Yaskawa INFORM job: A_ROOF_SIDE_0617_2_PAINT_21.JBI

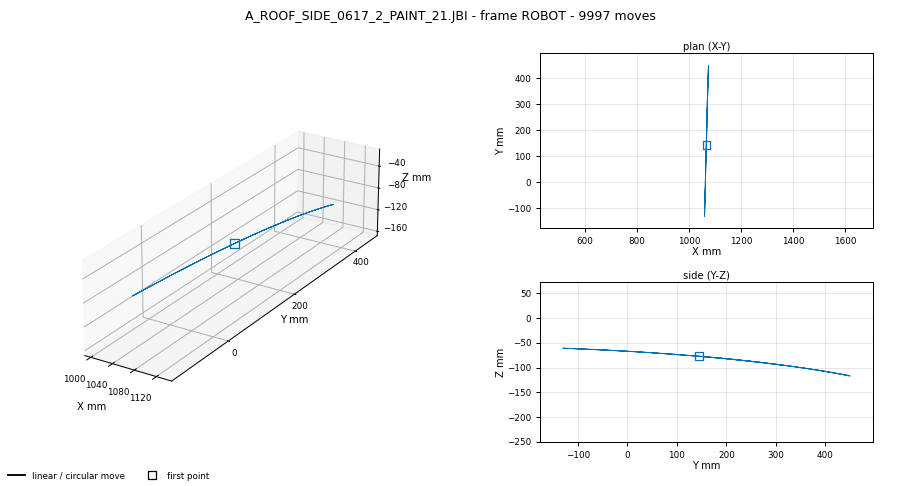
[picture p0: tool path of A_ROOF_SIDE_0617_2_PAINT_21.JBI in frame ROBOT, 9997 of 9997 moves have a stored position in this frame; points joined in program order, loops and branches not executed]
/JOB
//NAME A_ROOF_SIDE_0617_2_PAINT21
//POS
///NPOS 9997,0,0,0,0,0
///TOOL 1
///USER 0
///POSTYPE ROBOT
///RECTAN
///RCONF 1,0,0,0,0,0,0,0,0,0,0,0,0,0,0,0,0,0,0,0,0,0,0,0
C00000=1068.120,143.960,-76.437,172.975,27.840,155.057
C00001=1068.127,144.208,-76.458,172.976,27.843,155.058
C00002=1068.132,144.458,-76.479,172.978,27.845,155.058
C00003=1068.138,144.707,-76.500,172.981,27.848,155.058
C00004=1068.143,144.956,-76.521,172.982,27.851,155.059
C00005=1068.149,145.204,-76.542,172.984,27.854,155.059
C00006=1068.155,145.454,-76.563,172.985,27.857,155.059
C00007=1068.161,145.702,-76.584,172.988,27.860,155.060
C00008=1068.167,145.952,-76.605,172.989,27.862,155.060
C00009=1068.173,146.201,-76.626,172.991,27.865,155.061
C00010=1068.178,146.451,-76.647,172.992,27.868,155.061
C00011=1068.184,146.699,-76.668,172.995,27.870,155.061
C00012=1068.189,146.948,-76.689,172.996,27.873,155.062
C00013=1068.195,147.197,-76.710,172.998,27.876,155.062
C00014=1068.201,147.446,-76.730,172.999,27.879,155.063
C00015=1068.208,147.695,-76.752,173.001,27.881,155.063
C00016=1068.213,147.944,-76.773,173.003,27.885,155.063
C00017=1068.219,148.194,-76.794,173.005,27.887,155.064
C00018=1068.225,148.442,-76.816,173.007,27.890,155.064
C00019=1068.230,148.692,-76.836,173.008,27.893,155.065
C00020=1068.236,148.941,-76.858,173.011,27.896,155.065
C00021=1068.242,149.189,-76.879,173.012,27.898,155.065
C00022=1068.247,149.439,-76.900,173.014,27.901,155.066
C00023=1068.253,149.687,-76.921,173.015,27.904,155.066
C00024=1068.259,149.937,-76.943,173.018,27.907,155.066
C00025=1068.264,150.186,-76.963,173.019,27.909,155.067
C00026=1068.271,150.435,-76.985,173.021,27.912,155.067
C00027=1068.276,150.683,-77.006,173.022,27.915,155.068
C00028=1068.282,150.933,-77.028,173.025,27.918,155.068
C00029=1068.288,151.182,-77.048,173.026,27.921,155.068
C00030=1068.294,151.431,-77.070,173.028,27.923,155.069
C00031=1068.299,151.680,-77.092,173.030,27.926,155.069
C00032=1068.304,151.930,-77.113,173.032,27.929,155.070
C00033=1068.310,152.178,-77.134,173.034,27.932,155.070
C00034=1068.316,152.427,-77.156,173.035,27.935,155.070
C00035=1068.322,152.676,-77.177,173.038,27.938,155.071
C00036=1068.328,152.925,-77.199,173.039,27.940,155.071
C00037=1068.333,153.174,-77.219,173.041,27.943,155.071
C00038=1068.339,153.423,-77.241,173.042,27.945,155.072
C00039=1068.345,153.672,-77.262,173.045,27.948,155.072
C00040=1068.351,153.921,-77.284,173.046,27.951,155.073
C00041=1068.356,154.170,-77.306,173.048,27.954,155.073
C00042=1068.362,154.419,-77.327,173.049,27.957,155.074
C00043=1068.367,154.668,-77.348,173.052,27.960,155.074
C00044=1068.373,154.917,-77.369,173.053,27.962,155.074
C00045=1068.379,155.166,-77.391,173.055,27.965,155.075
C00046=1068.385,155.415,-77.412,173.058,27.968,155.075
C00047=1068.391,155.664,-77.434,173.059,27.971,155.075
C00048=1068.396,155.913,-77.456,173.061,27.974,155.076
C00049=1068.402,156.162,-77.478,173.062,27.976,155.076
C00050=1068.408,156.411,-77.499,173.065,27.979,155.077
C00051=1068.414,156.660,-77.520,173.066,27.982,155.077
C00052=1068.420,156.909,-77.542,173.068,27.985,155.078
C00053=1068.425,157.158,-77.564,173.070,27.988,155.078
C00054=1068.430,157.407,-77.584,173.072,27.990,155.078
C00055=1068.436,157.656,-77.606,173.073,27.993,155.079
C00056=1068.442,157.905,-77.627,173.076,27.996,155.079
C00057=1068.447,158.154,-77.650,173.077,27.999,155.079
C00058=1068.454,158.404,-77.671,173.079,28.001,155.080
C00059=1068.460,158.686,-77.696,173.081,28.005,155.080
C00060=1068.467,158.968,-77.721,173.083,28.008,155.081
C00061=1068.474,159.252,-77.745,173.085,28.011,155.081
C00062=1068.479,159.535,-77.770,173.088,28.014,155.082
C00063=1068.485,159.783,-77.792,173.089,28.017,155.082
C00064=1068.491,160.033,-77.813,173.091,28.020,155.082
C00065=1068.497,160.282,-77.835,173.094,28.023,155.083
C00066=1068.502,160.531,-77.857,173.095,28.025,155.083
C00067=1068.508,160.780,-77.878,173.097,28.028,155.084
C00068=1068.514,161.029,-77.900,173.099,28.031,155.084
C00069=1068.519,161.278,-77.922,173.101,28.034,155.084
C00070=1068.526,161.526,-77.944,173.102,28.037,155.085
C00071=1068.531,161.775,-77.966,173.104,28.039,155.085
C00072=1068.537,162.024,-77.988,173.106,28.042,155.086
C00073=1068.542,162.274,-78.010,173.108,28.045,155.086
C00074=1068.548,162.522,-78.031,173.109,28.048,155.086
C00075=1068.553,162.771,-78.054,173.112,28.051,155.087
C00076=1068.558,163.020,-78.076,173.113,28.054,155.087
C00077=1068.564,163.269,-78.098,173.115,28.057,155.088
C00078=1068.569,163.518,-78.120,173.117,28.060,155.088
C00079=1068.575,163.767,-78.141,173.119,28.063,155.088
C00080=1068.581,164.016,-78.164,173.121,28.065,155.089
C00081=1068.586,164.265,-78.186,173.123,28.068,155.089
C00082=1068.592,164.514,-78.208,173.125,28.071,155.090
C00083=1068.598,164.764,-78.230,173.126,28.074,155.090
C00084=1068.603,165.012,-78.252,173.129,28.077,155.090
C00085=1068.609,165.261,-78.274,173.130,28.080,155.091
C00086=1068.614,165.510,-78.296,173.132,28.083,155.091
C00087=1068.620,165.759,-78.318,173.134,28.086,155.092
C00088=1068.626,166.008,-78.340,173.136,28.089,155.092
C00089=1068.630,166.257,-78.362,173.138,28.092,155.093
C00090=1068.637,166.506,-78.385,173.140,28.094,155.093
C00091=1068.642,166.755,-78.407,173.141,28.097,155.093
C00092=1068.647,167.004,-78.429,173.144,28.100,155.094
C00093=1068.654,167.252,-78.451,173.145,28.103,155.094
C00094=1068.659,167.502,-78.473,173.147,28.106,155.095
C00095=1068.664,167.750,-78.496,173.150,28.109,155.095
C00096=1068.670,167.999,-78.518,173.151,28.112,155.096
C00097=1068.676,168.249,-78.540,173.153,28.115,155.096
C00098=1068.682,168.498,-78.562,173.155,28.118,155.096
C00099=1068.687,168.746,-78.584,173.157,28.120,155.097
C00100=1068.693,168.995,-78.607,173.159,28.123,155.097
C00101=1068.699,169.244,-78.629,173.161,28.126,155.098
C00102=1068.704,169.493,-78.651,173.162,28.129,155.098
C00103=1068.709,169.742,-78.673,173.165,28.132,155.098
C00104=1068.715,169.991,-78.696,173.166,28.135,155.099
C00105=1068.721,170.240,-78.718,173.168,28.137,155.099
C00106=1068.726,170.488,-78.741,173.170,28.140,155.100
C00107=1068.732,170.738,-78.763,173.172,28.143,155.100
C00108=1068.738,170.987,-78.785,173.175,28.146,155.100
C00109=1068.744,171.236,-78.807,173.176,28.149,155.101
C00110=1068.750,171.485,-78.830,173.178,28.151,155.101
C00111=1068.755,171.733,-78.852,173.180,28.155,155.102
C00112=1068.761,171.982,-78.875,173.182,28.158,155.102
C00113=1068.766,172.232,-78.897,173.184,28.161,155.102
C00114=1068.772,172.481,-78.920,173.186,28.163,155.103
C00115=1068.778,172.730,-78.941,173.187,28.166,155.103
C00116=1068.783,172.978,-78.964,173.190,28.169,155.104
C00117=1068.789,173.227,-78.987,173.191,28.172,155.104
C00118=1068.795,173.476,-79.009,173.194,28.175,155.104
C00119=1068.801,173.725,-79.031,173.195,28.178,155.105
C00120=1068.807,173.974,-79.054,173.197,28.180,155.105
C00121=1068.811,174.223,-79.076,173.200,28.183,155.106
C00122=1068.818,174.471,-79.099,173.201,28.186,155.106
C00123=1068.825,174.755,-79.125,173.204,28.190,155.107
C00124=1068.831,175.037,-79.150,173.206,28.193,155.107
C00125=1068.837,175.319,-79.175,173.208,28.196,155.107
C00126=1068.844,175.602,-79.201,173.210,28.199,155.108
C00127=1068.850,175.851,-79.224,173.213,28.202,155.108
C00128=1068.856,176.100,-79.246,173.214,28.205,155.109
C00129=1068.861,176.348,-79.269,173.217,28.208,155.109
C00130=1068.867,176.597,-79.292,173.218,28.210,155.109
C00131=1068.872,176.846,-79.314,173.220,28.213,155.110
C00132=1068.878,177.095,-79.336,173.222,28.216,155.110
C00133=1068.884,177.344,-79.359,173.224,28.219,155.111
C00134=1068.890,177.593,-79.382,173.226,28.222,155.111
C00135=1068.896,177.842,-79.405,173.228,28.225,155.112
C00136=1068.902,178.091,-79.427,173.230,28.228,155.112
C00137=1068.908,178.340,-79.450,173.232,28.231,155.112
C00138=1068.913,178.589,-79.472,173.235,28.234,155.113
C00139=1068.919,178.838,-79.495,173.236,28.236,155.113
C00140=1068.925,179.087,-79.518,173.239,28.239,155.113
C00141=1068.931,179.336,-79.541,173.240,28.242,155.114
C00142=1068.937,179.584,-79.564,173.242,28.245,155.114
C00143=1068.942,179.834,-79.586,173.244,28.248,155.115
C00144=1068.948,180.083,-79.609,173.246,28.251,155.115
C00145=1068.954,180.332,-79.632,173.248,28.254,155.115
C00146=1068.960,180.580,-79.654,173.250,28.256,155.116
C00147=1068.966,180.829,-79.677,173.252,28.259,155.116
C00148=1068.972,181.078,-79.700,173.254,28.262,155.117
C00149=1068.978,181.327,-79.723,173.257,28.265,155.117
C00150=1068.983,181.576,-79.746,173.258,28.268,155.117
C00151=1068.989,181.825,-79.769,173.261,28.271,155.118
C00152=1068.995,182.073,-79.791,173.262,28.273,155.118
C00153=1069.001,182.322,-79.814,173.265,28.276,155.119
C00154=1069.007,182.571,-79.837,173.266,28.279,155.119
C00155=1069.013,182.820,-79.860,173.269,28.282,155.119
C00156=1069.018,183.069,-79.883,173.270,28.285,155.120
C00157=1069.024,183.318,-79.906,173.273,28.288,155.120
C00158=1069.031,183.566,-79.928,173.275,28.290,155.121
C00159=1069.036,183.815,-79.951,173.277,28.293,155.121
C00160=1069.042,184.064,-79.974,173.279,28.296,155.121
C00161=1069.048,184.313,-79.997,173.281,28.299,155.122
C00162=1069.053,184.562,-80.020,173.283,28.302,155.122
C00163=1069.059,184.811,-80.043,173.285,28.305,155.123
C00164=1069.065,185.060,-80.066,173.287,28.307,155.123
C00165=1069.071,185.309,-80.089,173.289,28.310,155.123
C00166=1069.076,185.557,-80.113,173.291,28.314,155.124
C00167=1069.082,185.806,-80.136,173.293,28.317,155.124
C00168=1069.087,186.055,-80.159,173.295,28.319,155.125
C00169=1069.092,186.304,-80.183,173.298,28.322,155.125
C00170=1069.098,186.553,-80.206,173.299,28.326,155.126
C00171=1069.104,186.802,-80.229,173.302,28.329,155.126
C00172=1069.110,187.050,-80.252,173.303,28.331,155.126
C00173=1069.115,187.300,-80.276,173.306,28.335,155.127
C00174=1069.121,187.548,-80.299,173.307,28.338,155.127
C00175=1069.126,187.797,-80.322,173.310,28.341,155.128
C00176=1069.132,188.046,-80.346,173.311,28.343,155.128
C00177=1069.137,188.295,-80.369,173.314,28.347,155.129
C00178=1069.143,188.544,-80.392,173.315,28.350,155.129
C00179=1069.148,188.793,-80.415,173.318,28.352,155.130
C00180=1069.154,189.041,-80.439,173.319,28.355,155.130
C00181=1069.160,189.290,-80.462,173.322,28.359,155.130
C00182=1069.165,189.539,-80.485,173.324,28.362,155.131
C00183=1069.171,189.788,-80.509,173.326,28.364,155.131
C00184=1069.177,190.037,-80.532,173.329,28.367,155.132
C00185=1069.182,190.286,-80.556,173.330,28.371,155.132
C00186=1069.188,190.535,-80.580,173.333,28.374,155.133
C00187=1069.195,190.816,-80.606,173.335,28.377,155.133
C00188=1069.201,191.098,-80.632,173.337,28.380,155.134
C00189=1069.207,191.381,-80.660,173.339,28.384,155.134
C00190=1069.213,191.663,-80.686,173.342,28.387,155.134
C00191=1069.219,191.912,-80.709,173.344,28.390,155.135
C00192=1069.226,192.161,-80.733,173.346,28.393,155.135
C00193=1069.231,192.410,-80.757,173.348,28.396,155.136
C00194=1069.236,192.659,-80.780,173.351,28.399,155.136
C00195=1069.242,192.907,-80.804,173.352,28.402,155.137
C00196=1069.247,193.156,-80.827,173.355,28.405,155.137
C00197=1069.254,193.405,-80.850,173.356,28.408,155.137
C00198=1069.259,193.654,-80.874,173.359,28.411,155.138
C00199=1069.265,193.903,-80.898,173.360,28.414,155.138
C00200=1069.271,194.152,-80.921,173.363,28.417,155.139
C00201=1069.276,194.400,-80.945,173.365,28.420,155.139
C00202=1069.282,194.649,-80.968,173.367,28.423,155.140
C00203=1069.287,194.898,-80.992,173.370,28.426,155.140
C00204=1069.293,195.146,-81.016,173.371,28.429,155.141
C00205=1069.300,195.396,-81.039,173.374,28.432,155.141
C00206=1069.305,195.644,-81.064,173.376,28.435,155.141
C00207=1069.311,195.893,-81.087,173.378,28.438,155.142
C00208=1069.316,196.142,-81.111,173.380,28.441,155.142
C00209=1069.322,196.391,-81.134,173.382,28.444,155.143
C00210=1069.328,196.640,-81.158,173.384,28.447,155.143
C00211=1069.334,196.888,-81.182,173.387,28.450,155.144
C00212=1069.339,197.137,-81.205,173.388,28.453,155.144
C00213=1069.345,197.386,-81.230,173.391,28.456,155.144
C00214=1069.351,197.635,-81.253,173.393,28.459,155.145
C00215=1069.356,197.884,-81.277,173.395,28.462,155.145
C00216=1069.362,198.132,-81.300,173.398,28.465,155.146
C00217=1069.368,198.381,-81.325,173.399,28.468,155.146
C00218=1069.374,198.630,-81.349,173.402,28.471,155.147
C00219=1069.380,198.879,-81.372,173.403,28.474,155.147
C00220=1069.385,199.127,-81.396,173.406,28.477,155.147
C00221=1069.392,199.376,-81.420,173.408,28.481,155.148
C00222=1069.397,199.625,-81.444,173.410,28.483,155.148
C00223=1069.403,199.874,-81.467,173.412,28.486,155.149
C00224=1069.409,200.123,-81.492,173.415,28.489,155.149
C00225=1069.415,200.371,-81.515,173.416,28.492,155.150
C00226=1069.420,200.620,-81.540,173.419,28.495,155.150
C00227=1069.426,200.869,-81.563,173.422,28.498,155.150
C00228=1069.432,201.118,-81.587,173.423,28.501,155.151
C00229=1069.438,201.366,-81.611,173.426,28.504,155.151
C00230=1069.444,201.616,-81.636,173.428,28.507,155.152
C00231=1069.450,201.864,-81.659,173.430,28.510,155.152
C00232=1069.455,202.112,-81.683,173.432,28.513,155.152
C00233=1069.461,202.362,-81.707,173.434,28.516,155.153
C00234=1069.467,202.611,-81.731,173.436,28.519,155.153
C00235=1069.472,202.859,-81.755,173.439,28.523,155.154
C00236=1069.479,203.108,-81.779,173.441,28.525,155.154
C00237=1069.484,203.357,-81.804,173.443,28.528,155.155
C00238=1069.489,203.605,-81.828,173.446,28.532,155.155
C00239=1069.494,203.826,-81.850,173.447,28.535,155.156
C00240=1069.500,204.046,-81.871,173.449,28.537,155.156
C00241=1069.504,204.268,-81.892,173.451,28.540,155.156
C00242=1069.509,204.488,-81.914,173.453,28.543,155.157
C00243=1069.514,204.709,-81.935,173.455,28.546,155.157
C00244=1069.520,204.929,-81.957,173.457,28.549,155.158
C00245=1069.525,205.150,-81.978,173.459,28.551,155.158
C00246=1069.530,205.371,-82.000,173.461,28.554,155.158
C00247=1069.535,205.619,-82.024,173.463,28.557,155.159
C00248=1069.542,205.868,-82.048,173.465,28.560,155.159
C00249=1069.547,206.117,-82.073,173.468,28.563,155.160
C00250=1069.553,206.366,-82.097,173.469,28.566,155.160
C00251=1069.581,207.634,-82.221,173.612,28.641,155.164
C00252=1069.587,207.847,-82.243,173.614,28.644,155.164
C00253=1069.592,208.061,-82.265,173.616,28.648,155.165
C00254=1069.598,208.275,-82.286,173.618,28.651,155.165
C00255=1069.602,208.489,-82.308,173.619,28.655,155.166
C00256=1069.608,208.703,-82.329,173.621,28.658,155.167
C00257=1069.612,208.917,-82.351,173.622,28.662,155.167
C00258=1069.617,209.131,-82.373,173.625,28.665,155.168
C00259=1069.623,209.344,-82.394,173.626,28.668,155.168
C00260=1069.629,209.593,-82.419,173.629,28.673,155.169
C00261=1069.634,209.841,-82.444,173.630,28.677,155.170
C00262=1069.640,210.090,-82.469,173.633,28.681,155.170
C00263=1069.646,210.339,-82.495,173.634,28.685,155.171
C00264=1069.652,210.588,-82.520,173.636,28.689,155.171
C00265=1069.658,210.836,-82.545,173.639,28.693,155.172
C00266=1069.664,211.084,-82.570,173.640,28.697,155.173
C00267=1069.670,211.334,-82.595,173.643,28.701,155.173
C00268=1069.675,211.583,-82.621,173.644,28.705,155.174
C00269=1069.681,211.831,-82.646,173.647,28.709,155.175
C00270=1069.687,212.079,-82.671,173.649,28.713,155.175
C00271=1069.693,212.328,-82.697,173.650,28.717,155.176
C00272=1069.699,212.576,-82.722,173.653,28.721,155.177
C00273=1069.705,212.825,-82.748,173.654,28.725,155.178
C00274=1069.711,213.074,-82.773,173.657,28.729,155.178
C00275=1069.717,213.322,-82.798,173.659,28.733,155.179
C00276=1069.722,213.571,-82.824,173.661,28.737,155.179
C00277=1069.728,213.820,-82.849,173.663,28.741,155.180
C00278=1069.735,214.068,-82.875,173.665,28.745,155.181
C00279=1069.739,214.317,-82.900,173.667,28.749,155.181
C00280=1069.746,214.565,-82.926,173.669,28.753,155.182
C00281=1069.752,214.814,-82.951,173.671,28.757,155.183
C00282=1069.757,215.063,-82.977,173.673,28.761,155.183
C00283=1069.764,215.312,-83.002,173.676,28.765,155.184
C00284=1069.769,215.561,-83.028,173.677,28.769,155.185
C00285=1069.775,215.809,-83.053,173.679,28.773,155.185
C00286=1069.781,216.057,-83.078,173.682,28.777,155.186
C00287=1069.786,216.306,-83.104,173.683,28.781,155.187
C00288=1069.792,216.555,-83.130,173.686,28.785,155.187
C00289=1069.799,216.804,-83.155,173.687,28.789,155.188
C00290=1069.804,217.053,-83.181,173.690,28.793,155.189
C00291=1069.810,217.301,-83.206,173.692,28.797,155.189
C00292=1069.815,217.550,-83.232,173.694,28.801,155.190
C00293=1069.822,217.798,-83.258,173.696,28.805,155.191
C00294=1069.828,218.046,-83.283,173.698,28.809,155.191
C00295=1069.833,218.295,-83.309,173.700,28.813,155.192
C00296=1069.840,218.544,-83.335,173.702,28.817,155.193
C00297=1069.845,218.793,-83.361,173.705,28.821,155.193
C00298=1069.852,219.041,-83.387,173.706,28.825,155.194
C00299=1069.857,219.290,-83.413,173.709,28.829,155.195
C00300=1069.863,219.539,-83.438,173.711,28.833,155.195
C00301=1069.869,219.787,-83.463,173.713,28.837,155.196
C00302=1069.875,220.036,-83.490,173.715,28.841,155.197
C00303=1069.881,220.284,-83.515,173.717,28.845,155.197
C00304=1069.887,220.533,-83.541,173.719,28.849,155.198
C00305=1069.893,220.782,-83.566,173.721,28.853,155.199
C00306=1069.899,221.030,-83.593,173.724,28.857,155.199
C00307=1069.905,221.279,-83.618,173.725,28.861,155.200
C00308=1069.910,221.495,-83.641,173.728,28.864,155.200
C00309=1069.915,221.711,-83.663,173.729,28.868,155.201
C00310=1069.920,221.927,-83.686,173.731,28.871,155.202
C00311=1069.925,222.143,-83.709,173.733,28.875,155.202
C00312=1069.930,222.359,-83.732,173.735,28.878,155.203
C00313=1069.936,222.575,-83.754,173.736,28.882,155.203
C00314=1069.940,222.791,-83.776,173.739,28.885,155.204
C00315=1069.945,223.007,-83.799,173.740,28.889,155.205
C00316=1069.951,223.255,-83.825,173.743,28.893,155.205
C00317=1069.957,223.504,-83.851,173.744,28.897,155.206
C00318=1069.963,223.752,-83.877,173.747,28.901,155.207
C00319=1069.969,224.001,-83.903,173.749,28.905,155.207
C00320=1069.974,224.250,-83.930,173.751,28.908,155.208
C00321=1069.981,224.498,-83.955,173.753,28.912,155.208
C00322=1069.986,224.747,-83.982,173.756,28.916,155.209
C00323=1069.992,224.996,-84.008,173.757,28.921,155.210
C00324=1069.998,225.244,-84.034,173.760,28.925,155.211
C00325=1070.004,225.493,-84.060,173.762,28.929,155.211
C00326=1070.010,225.741,-84.086,173.764,28.933,155.212
C00327=1070.016,225.990,-84.112,173.766,28.936,155.212
C00328=1070.022,226.238,-84.138,173.768,28.940,155.213
C00329=1070.027,226.487,-84.164,173.771,28.944,155.214
C00330=1070.033,226.735,-84.191,173.772,28.948,155.214
C00331=1070.039,226.983,-84.217,173.775,28.952,155.215
C00332=1070.045,227.233,-84.243,173.777,28.956,155.216
C00333=1070.051,227.481,-84.270,173.780,28.960,155.216
C00334=1070.057,227.730,-84.297,173.781,28.964,155.217
C00335=1070.063,227.978,-84.322,173.784,28.968,155.218
C00336=1070.069,228.227,-84.349,173.786,28.972,155.218
C00337=1070.075,228.475,-84.375,173.789,28.976,155.219
C00338=1070.081,228.724,-84.401,173.790,28.980,155.220
C00339=1070.087,228.972,-84.427,173.793,28.984,155.220
C00340=1070.093,229.221,-84.454,173.795,28.987,155.221
C00341=1070.098,229.470,-84.480,173.796,28.991,155.221
C00342=1070.104,229.719,-84.507,173.799,28.995,155.222
C00343=1070.111,229.967,-84.533,173.801,29.000,155.223
C00344=1070.117,230.215,-84.559,173.804,29.004,155.224
C00345=1070.122,230.464,-84.585,173.805,29.008,155.224
C00346=1070.128,230.712,-84.612,173.808,29.011,155.225
C00347=1070.134,230.961,-84.639,173.810,29.015,155.225
C00348=1070.140,231.210,-84.666,173.813,29.019,155.226
C00349=1070.146,231.458,-84.692,173.814,29.023,155.227
C00350=1070.151,231.707,-84.719,173.817,29.027,155.227
C00351=1070.157,231.956,-84.745,173.819,29.031,155.228
C00352=1070.163,232.204,-84.772,173.822,29.035,155.229
C00353=1070.168,232.452,-84.798,173.823,29.039,155.229
C00354=1070.175,232.701,-84.825,173.826,29.043,155.230
C00355=1070.181,232.950,-84.852,173.828,29.047,155.231
C00356=1070.186,233.198,-84.879,173.830,29.051,155.231
C00357=1070.192,233.446,-84.905,173.832,29.055,155.232
C00358=1070.198,233.695,-84.932,173.834,29.059,155.233
C00359=1070.204,233.943,-84.959,173.837,29.063,155.233
C00360=1070.210,234.192,-84.986,173.839,29.067,155.234
C00361=1070.216,234.441,-85.012,173.841,29.071,155.235
C00362=1070.222,234.689,-85.039,173.843,29.075,155.235
C00363=1070.227,234.937,-85.065,173.846,29.079,155.236
C00364=1070.232,235.149,-85.088,173.847,29.082,155.236
C00365=1070.238,235.361,-85.112,173.850,29.086,155.237
C00366=1070.242,235.573,-85.135,173.851,29.089,155.238
C00367=1070.247,235.785,-85.156,173.853,29.092,155.238
C00368=1070.252,235.997,-85.179,173.856,29.096,155.239
C00369=1070.258,236.210,-85.203,173.857,29.099,155.239
C00370=1070.262,236.421,-85.226,173.860,29.102,155.240
C00371=1070.267,236.633,-85.249,173.861,29.106,155.240
C00372=1070.273,236.882,-85.275,173.864,29.110,155.241
C00373=1070.280,237.130,-85.303,173.866,29.114,155.242
C00374=1070.285,237.378,-85.330,173.868,29.118,155.242
C00375=1070.291,237.627,-85.356,173.870,29.122,155.243
C00376=1070.298,237.876,-85.383,173.873,29.126,155.244
C00377=1070.303,238.124,-85.410,173.875,29.130,155.244
C00378=1070.308,238.373,-85.437,173.878,29.134,155.245
C00379=1070.314,238.621,-85.464,173.879,29.137,155.246
C00380=1070.321,238.870,-85.491,173.882,29.141,155.246
C00381=1070.327,239.118,-85.518,173.884,29.145,155.247
C00382=1070.332,239.366,-85.545,173.887,29.149,155.248
C00383=1070.339,239.615,-85.572,173.889,29.153,155.248
C00384=1070.344,239.863,-85.600,173.891,29.157,155.249
C00385=1070.350,240.112,-85.626,173.893,29.161,155.250
C00386=1070.356,240.361,-85.653,173.896,29.165,155.250
C00387=1070.362,240.609,-85.681,173.898,29.169,155.251
C00388=1070.367,240.857,-85.708,173.901,29.173,155.251
C00389=1070.374,241.106,-85.735,173.902,29.177,155.252
C00390=1070.380,241.354,-85.762,173.905,29.181,155.253
C00391=1070.386,241.602,-85.789,173.907,29.185,155.253
C00392=1070.392,241.851,-85.816,173.910,29.189,155.254
C00393=1070.397,242.100,-85.844,173.912,29.192,155.255
C00394=1070.404,242.349,-85.871,173.915,29.196,155.255
C00395=1070.410,242.596,-85.898,173.916,29.200,155.256
C00396=1070.415,242.845,-85.926,173.919,29.204,155.257
C00397=1070.421,243.093,-85.953,173.921,29.208,155.257
C00398=1070.427,243.342,-85.980,173.923,29.213,155.258
C00399=1070.432,243.590,-86.007,173.926,29.217,155.259
C00400=1070.439,243.839,-86.035,173.928,29.221,155.259
C00401=1070.444,244.088,-86.062,173.930,29.224,155.260
C00402=1070.451,244.336,-86.090,173.932,29.228,155.261
C00403=1070.456,244.584,-86.118,173.935,29.232,155.261
C00404=1070.462,244.832,-86.145,173.937,29.236,155.262
C00405=1070.468,245.081,-86.172,173.940,29.240,155.263
C00406=1070.473,245.330,-86.200,173.942,29.244,155.263
C00407=1070.480,245.578,-86.227,173.945,29.248,155.264
C00408=1070.485,245.827,-86.255,173.946,29.252,155.265
C00409=1070.491,246.074,-86.282,173.949,29.256,155.265
C00410=1070.497,246.323,-86.310,173.951,29.260,155.266
C00411=1070.503,246.572,-86.337,173.954,29.264,155.266
C00412=1070.509,246.820,-86.365,173.956,29.268,155.267
C00413=1070.515,247.068,-86.393,173.959,29.272,155.268
C00414=1070.521,247.317,-86.420,173.961,29.276,155.269
C00415=1070.526,247.565,-86.448,173.963,29.280,155.269
C00416=1070.532,247.813,-86.475,173.965,29.284,155.270
C00417=1070.538,248.063,-86.503,173.968,29.288,155.271
C00418=1070.543,248.311,-86.531,173.970,29.292,155.271
C00419=1070.550,248.559,-86.559,173.973,29.296,155.272
C00420=1070.559,248.977,-86.605,173.977,29.303,155.273
C00421=1070.569,249.394,-86.652,173.981,29.309,155.274
C00422=1070.579,249.811,-86.698,173.984,29.316,155.275
C00423=1070.588,250.229,-86.746,173.989,29.323,155.276
C00424=1070.594,250.477,-86.774,173.991,29.327,155.277
C00425=1070.600,250.725,-86.802,173.994,29.331,155.278
C00426=1070.605,250.974,-86.829,173.996,29.334,155.278
C00427=1070.611,251.223,-86.857,173.999,29.338,155.279
C00428=1070.617,251.470,-86.884,174.001,29.343,155.280
C00429=1070.623,251.719,-86.913,174.004,29.347,155.280
C00430=1070.629,251.967,-86.941,174.005,29.351,155.281
C00431=1070.635,252.216,-86.969,174.008,29.355,155.282
C00432=1070.641,252.464,-86.996,174.010,29.358,155.282
C00433=1070.647,252.712,-87.025,174.013,29.362,155.283
C00434=1070.652,252.961,-87.053,174.015,29.366,155.284
C00435=1070.658,253.209,-87.081,174.018,29.370,155.284
C00436=1070.664,253.458,-87.109,174.020,29.374,155.285
C00437=1070.670,253.706,-87.137,174.023,29.378,155.286
C00438=1070.676,253.954,-87.165,174.025,29.382,155.286
C00439=1070.681,254.202,-87.193,174.028,29.387,155.287
C00440=1070.688,254.451,-87.221,174.030,29.390,155.288
C00441=1070.694,254.700,-87.249,174.033,29.394,155.288
C00442=1070.699,254.948,-87.277,174.034,29.398,155.289
C00443=1070.705,255.196,-87.305,174.037,29.402,155.290
C00444=1070.711,255.444,-87.333,174.039,29.406,155.290
C00445=1070.717,255.692,-87.362,174.042,29.410,155.291
C00446=1070.723,255.941,-87.390,174.044,29.414,155.292
C00447=1070.729,256.189,-87.418,174.047,29.418,155.292
C00448=1070.735,256.438,-87.446,174.049,29.422,155.293
C00449=1070.741,256.686,-87.474,174.052,29.426,155.293
C00450=1070.747,256.934,-87.502,174.054,29.430,155.294
C00451=1070.753,257.182,-87.531,174.057,29.434,155.295
C00452=1070.759,257.431,-87.559,174.059,29.437,155.295
C00453=1070.764,257.679,-87.587,174.062,29.441,155.296
C00454=1070.771,257.928,-87.615,174.065,29.445,155.297
C00455=1070.777,258.176,-87.644,174.067,29.449,155.297
C00456=1070.783,258.425,-87.672,174.070,29.453,155.298
C00457=1070.788,258.673,-87.700,174.072,29.457,155.299
C00458=1070.794,258.921,-87.729,174.075,29.461,155.299
C00459=1070.801,259.170,-87.758,174.077,29.465,155.300
C00460=1070.807,259.418,-87.786,174.080,29.469,155.301
C00461=1070.813,259.666,-87.813,174.082,29.473,155.301
C00462=1070.819,259.914,-87.843,174.085,29.477,155.302
C00463=1070.825,260.163,-87.871,174.087,29.481,155.303
C00464=1070.831,260.411,-87.900,174.089,29.484,155.303
C00465=1070.836,260.659,-87.928,174.091,29.488,155.304
C00466=1070.843,260.908,-87.956,174.094,29.492,155.305
C00467=1070.849,261.156,-87.985,174.096,29.496,155.305
C00468=1070.855,261.404,-88.013,174.099,29.500,155.306
C00469=1070.861,261.653,-88.042,174.101,29.504,155.306
C00470=1070.867,261.901,-88.070,174.104,29.508,155.307
C00471=1070.873,262.149,-88.099,174.107,29.512,155.308
C00472=1070.883,262.564,-88.146,174.111,29.518,155.309
C00473=1070.893,262.979,-88.194,174.115,29.525,155.310
C00474=1070.903,263.394,-88.242,174.119,29.531,155.311
C00475=1070.913,263.809,-88.290,174.123,29.538,155.312
C00476=1070.920,264.057,-88.319,174.126,29.542,155.313
C00477=1070.926,264.306,-88.347,174.128,29.546,155.314
C00478=1070.931,264.554,-88.376,174.131,29.550,155.314
C00479=1070.937,264.802,-88.405,174.134,29.554,155.315
C00480=1070.943,265.050,-88.433,174.137,29.558,155.315
C00481=1070.949,265.299,-88.463,174.140,29.562,155.316
C00482=1070.955,265.547,-88.492,174.142,29.566,155.317
C00483=1070.961,265.795,-88.520,174.145,29.570,155.318
C00484=1070.967,266.043,-88.549,174.147,29.574,155.318
C00485=1070.973,266.291,-88.578,174.150,29.578,155.319
C00486=1070.979,266.540,-88.608,174.152,29.582,155.319
C00487=1070.984,266.789,-88.636,174.155,29.586,155.320
C00488=1070.991,267.037,-88.665,174.157,29.590,155.321
C00489=1070.997,267.285,-88.694,174.160,29.594,155.321
C00490=1071.003,267.532,-88.723,174.162,29.598,155.322
C00491=1071.008,267.781,-88.752,174.165,29.602,155.323
C00492=1071.014,268.029,-88.781,174.167,29.606,155.323
C00493=1071.020,268.278,-88.810,174.170,29.610,155.324
C00494=1071.027,268.526,-88.839,174.173,29.614,155.325
C00495=1071.032,268.774,-88.868,174.175,29.618,155.325
C00496=1071.038,269.022,-88.897,174.178,29.622,155.326
C00497=1071.045,269.270,-88.926,174.180,29.626,155.327
C00498=1071.050,269.519,-88.956,174.183,29.630,155.327
C00499=1071.056,269.768,-88.984,174.185,29.634,155.328
C00500=1071.062,270.015,-89.013,174.188,29.638,155.329
C00501=1071.067,270.263,-89.043,174.190,29.642,155.329
C00502=1071.073,270.512,-89.072,174.193,29.646,155.330
C00503=1071.080,270.760,-89.101,174.195,29.650,155.331
C00504=1071.085,271.008,-89.130,174.198,29.654,155.332
C00505=1071.091,271.256,-89.159,174.200,29.658,155.332
C00506=1071.098,271.504,-89.188,174.203,29.662,155.333
C00507=1071.103,271.753,-89.218,174.207,29.666,155.333
C00508=1071.109,272.001,-89.247,174.209,29.670,155.334
C00509=1071.115,272.249,-89.277,174.212,29.674,155.335
C00510=1071.122,272.497,-89.307,174.214,29.678,155.336
C00511=1071.128,272.745,-89.336,174.217,29.682,155.336
C00512=1071.133,272.993,-89.365,174.219,29.686,155.337
C00513=1071.140,273.242,-89.394,174.222,29.690,155.338
C00514=1071.145,273.490,-89.424,174.224,29.694,155.338
C00515=1071.151,273.738,-89.453,174.227,29.698,155.339
C00516=1071.157,273.987,-89.483,174.229,29.702,155.340
C00517=1071.163,274.234,-89.512,174.232,29.706,155.340
C00518=1071.169,274.483,-89.542,174.235,29.710,155.341
C00519=1071.175,274.731,-89.571,174.237,29.714,155.342
C00520=1071.181,274.979,-89.601,174.241,29.719,155.342
C00521=1071.186,275.228,-89.630,174.243,29.722,155.343
C00522=1071.193,275.475,-89.660,174.246,29.726,155.344
C00523=1071.198,275.724,-89.690,174.248,29.730,155.344
C00524=1071.208,276.142,-89.739,174.252,29.737,155.346
C00525=1071.219,276.560,-89.789,174.257,29.744,155.347
C00526=1071.228,276.978,-89.839,174.262,29.751,155.348
C00527=1071.238,277.397,-89.889,174.266,29.758,155.349
C00528=1071.244,277.645,-89.919,174.269,29.762,155.350
C00529=1071.250,277.893,-89.949,174.271,29.766,155.350
C00530=1071.257,278.141,-89.979,174.274,29.770,155.351
C00531=1071.262,278.390,-90.009,174.276,29.774,155.352
C00532=1071.268,278.638,-90.038,174.279,29.778,155.352
C00533=1071.275,278.886,-90.068,174.282,29.782,155.353
C00534=1071.280,279.134,-90.098,174.285,29.786,155.354
C00535=1071.286,279.382,-90.128,174.288,29.790,155.354
C00536=1071.292,279.630,-90.157,174.290,29.794,155.355
C00537=1071.298,279.878,-90.187,174.293,29.798,155.356
C00538=1071.304,280.127,-90.217,174.295,29.802,155.356
C00539=1071.311,280.374,-90.247,174.298,29.806,155.357
C00540=1071.316,280.623,-90.277,174.300,29.810,155.358
C00541=1071.322,280.871,-90.307,174.304,29.814,155.358
C00542=1071.328,281.119,-90.337,174.306,29.819,155.359
C00543=1071.333,281.367,-90.367,174.309,29.823,155.360
C00544=1071.340,281.614,-90.397,174.312,29.826,155.361
C00545=1071.346,281.862,-90.427,174.314,29.831,155.361
C00546=1071.352,282.111,-90.457,174.317,29.835,155.362
C00547=1071.358,282.359,-90.488,174.319,29.839,155.363
C00548=1071.363,282.607,-90.518,174.323,29.843,155.363
C00549=1071.369,282.856,-90.548,174.325,29.847,155.364
C00550=1071.375,283.103,-90.578,174.328,29.851,155.365
C00551=1071.381,283.351,-90.608,174.330,29.855,155.366
C00552=1071.387,283.600,-90.638,174.333,29.859,155.366
C00553=1071.393,283.848,-90.668,174.336,29.864,155.367
C00554=1071.399,284.096,-90.698,174.339,29.868,155.368
C00555=1071.405,284.343,-90.729,174.342,29.872,155.368
C00556=1071.411,284.591,-90.759,174.344,29.876,155.369
C00557=1071.417,284.840,-90.789,174.347,29.880,155.370
C00558=1071.423,285.088,-90.819,174.349,29.884,155.370
C00559=1071.428,285.336,-90.850,174.353,29.888,155.371
C00560=1071.434,285.584,-90.880,174.355,29.892,155.372
C00561=1071.441,285.832,-90.911,174.358,29.896,155.372
C00562=1071.446,286.080,-90.941,174.361,29.901,155.373
C00563=1071.453,286.328,-90.971,174.363,29.904,155.374
C00564=1071.459,286.577,-91.001,174.366,29.909,155.375
C00565=1071.465,286.825,-91.031,174.369,29.913,155.375
C00566=1071.471,287.073,-91.062,174.372,29.917,155.376
C00567=1071.477,287.320,-91.092,174.374,29.921,155.377
C00568=1071.483,287.569,-91.123,174.377,29.925,155.377
C00569=1071.489,287.817,-91.153,174.380,29.929,155.378
C00570=1071.495,288.065,-91.183,174.383,29.934,155.379
C00571=1071.501,288.313,-91.214,174.386,29.937,155.379
C00572=1071.507,288.561,-91.244,174.388,29.941,155.380
C00573=1071.513,288.809,-91.275,174.391,29.946,155.381
C00574=1071.519,289.057,-91.305,174.394,29.950,155.382
C00575=1071.525,289.305,-91.336,174.397,29.954,155.382
C00576=1071.530,289.519,-91.363,174.400,29.957,155.383
C00577=1071.536,289.733,-91.389,174.401,29.961,155.384
C00578=1071.541,289.948,-91.416,174.404,29.965,155.384
C00579=1071.545,290.162,-91.443,174.406,29.968,155.385
C00580=1071.551,290.376,-91.469,174.409,29.972,155.385
C00581=1071.556,290.591,-91.495,174.411,29.975,155.386
C00582=1071.561,290.805,-91.521,174.413,29.979,155.387
C00583=1071.566,291.019,-91.548,174.416,29.982,155.387
C00584=1071.572,291.267,-91.579,174.419,29.987,155.388
C00585=1071.578,291.514,-91.610,174.422,29.991,155.389
C00586=1071.585,291.763,-91.640,174.425,29.995,155.389
C00587=1071.590,292.011,-91.671,174.427,29.999,155.390
C00588=1071.596,292.259,-91.702,174.430,30.003,155.391
C00589=1071.602,292.507,-91.733,174.433,30.008,155.391
C00590=1071.608,292.755,-91.764,174.436,30.012,155.392
C00591=1071.614,293.004,-91.795,174.438,30.016,155.393
C00592=1071.620,293.251,-91.826,174.441,30.020,155.394
C00593=1071.626,293.499,-91.856,174.445,30.025,155.394
C00594=1071.632,293.747,-91.887,174.447,30.029,155.395
C00595=1071.638,293.995,-91.919,174.450,30.033,155.396
C00596=1071.644,294.243,-91.949,174.452,30.037,155.396
C00597=1071.650,294.490,-91.980,174.456,30.041,155.397
C00598=1071.657,294.739,-92.011,174.458,30.045,155.398
C00599=1071.662,294.987,-92.042,174.461,30.050,155.399
C00600=1071.668,295.235,-92.073,174.464,30.053,155.399
C00601=1071.674,295.483,-92.104,174.467,30.058,155.400
C00602=1071.681,295.731,-92.135,174.470,30.062,155.401
C00603=1071.686,295.979,-92.166,174.472,30.066,155.402
C00604=1071.692,296.226,-92.197,174.476,30.071,155.402
C00605=1071.698,296.475,-92.229,174.478,30.075,155.403
C00606=1071.704,296.722,-92.260,174.481,30.079,155.404
C00607=1071.711,296.970,-92.291,174.484,30.083,155.404
C00608=1071.716,297.218,-92.322,174.487,30.088,155.405
C00609=1071.723,297.466,-92.353,174.490,30.092,155.406
C00610=1071.728,297.714,-92.384,174.492,30.096,155.407
C00611=1071.734,297.962,-92.416,174.496,30.100,155.407
C00612=1071.740,298.209,-92.448,174.498,30.105,155.408
C00613=1071.745,298.458,-92.479,174.501,30.109,155.409
C00614=1071.751,298.705,-92.510,174.505,30.114,155.410
C00615=1071.757,298.954,-92.542,174.507,30.117,155.410
C00616=1071.763,299.201,-92.572,174.510,30.122,155.411
C00617=1071.769,299.450,-92.604,174.512,30.126,155.412
C00618=1071.775,299.697,-92.636,174.516,30.131,155.413
C00619=1071.781,299.945,-92.667,174.518,30.135,155.413
C00620=1071.787,300.193,-92.699,174.521,30.139,155.414
C00621=1071.792,300.441,-92.730,174.525,30.144,155.415
C00622=1071.799,300.689,-92.761,174.527,30.148,155.416
C00623=1071.805,300.937,-92.793,174.530,30.152,155.417
C00624=1071.810,301.184,-92.825,174.533,30.156,155.417
C00625=1071.817,301.432,-92.857,174.536,30.161,155.418
C00626=1071.823,301.681,-92.889,174.538,30.165,155.419
C00627=1071.828,301.929,-92.920,174.542,30.170,155.419
C00628=1071.834,302.177,-92.951,174.545,30.174,155.420
C00629=1071.840,302.424,-92.983,174.547,30.178,155.421
C00630=1071.846,302.672,-93.015,174.551,30.182,155.422
C00631=1071.852,302.919,-93.046,174.553,30.187,155.422
C00632=1071.858,303.141,-93.074,174.556,30.191,155.423
C00633=1071.863,303.363,-93.103,174.559,30.194,155.424
C00634=1071.868,303.584,-93.131,174.561,30.199,155.425
C00635=1071.874,303.806,-93.160,174.564,30.203,155.425
C00636=1071.879,304.028,-93.188,174.566,30.206,155.426
C00637=1071.884,304.249,-93.217,174.569,30.210,155.427
C00638=1071.889,304.472,-93.245,174.572,30.214,155.427
C00639=1071.894,304.693,-93.273,174.574,30.218,155.428
C00640=1071.901,304.941,-93.305,174.577,30.222,155.429
C00641=1071.907,305.188,-93.337,174.580,30.227,155.429
C00642=1071.913,305.436,-93.369,174.583,30.231,155.430
C00643=1071.919,305.684,-93.401,174.587,30.235,155.431
C00644=1071.925,305.932,-93.433,174.589,30.240,155.432
C00645=1071.931,306.179,-93.464,174.592,30.244,155.432
C00646=1071.937,306.428,-93.496,174.595,30.248,155.433
C00647=1071.943,306.676,-93.528,174.598,30.253,155.434
C00648=1071.949,306.922,-93.560,174.602,30.257,155.435
C00649=1071.955,307.171,-93.592,174.604,30.262,155.436
C00650=1071.961,307.419,-93.624,174.607,30.266,155.436
C00651=1071.967,307.667,-93.656,174.610,30.270,155.437
C00652=1071.974,307.914,-93.688,174.613,30.274,155.438
C00653=1071.980,308.162,-93.720,174.617,30.279,155.439
C00654=1071.986,308.410,-93.752,174.619,30.283,155.439
C00655=1071.992,308.658,-93.784,174.622,30.288,155.440
C00656=1071.998,308.906,-93.817,174.625,30.292,155.441
C00657=1072.004,309.153,-93.848,174.628,30.297,155.442
C00658=1072.010,309.401,-93.881,174.631,30.301,155.442
C00659=1072.016,309.649,-93.913,174.634,30.305,155.443
C00660=1072.022,309.897,-93.945,174.638,30.309,155.444
C00661=1072.029,310.145,-93.977,174.640,30.314,155.445
C00662=1072.035,310.393,-94.009,174.643,30.318,155.446
C00663=1072.041,310.641,-94.041,174.646,30.323,155.446
C00664=1072.048,310.888,-94.074,174.649,30.327,155.447
C00665=1072.053,311.136,-94.105,174.653,30.332,155.448
C00666=1072.059,311.384,-94.138,174.655,30.336,155.449
C00667=1072.065,311.632,-94.170,174.659,30.340,155.449
C00668=1072.071,311.879,-94.203,174.661,30.345,155.450
C00669=1072.077,312.128,-94.235,174.665,30.349,155.451
C00670=1072.084,312.375,-94.267,174.668,30.354,155.452
C00671=1072.090,312.623,-94.299,174.670,30.358,155.453
C00672=1072.097,312.871,-94.332,174.674,30.363,155.453
C00673=1072.103,313.118,-94.364,174.676,30.367,155.454
C00674=1072.109,313.366,-94.396,174.680,30.371,155.455
C00675=1072.115,313.614,-94.429,174.683,30.376,155.456
C00676=1072.121,313.862,-94.461,174.686,30.380,155.456
C00677=1072.128,314.110,-94.494,174.689,30.385,155.457
C00678=1072.134,314.357,-94.527,174.692,30.389,155.458
C00679=1072.140,314.606,-94.559,174.695,30.393,155.459
C00680=1072.146,314.853,-94.591,174.698,30.398,155.460
C00681=1072.152,315.101,-94.625,174.701,30.402,155.460
C00682=1072.158,315.349,-94.658,174.705,30.407,155.461
C00683=1072.163,315.596,-94.689,174.707,30.412,155.462
C00684=1072.169,315.844,-94.723,174.710,30.416,155.463
C00685=1072.175,316.092,-94.755,174.713,30.421,155.464
C00686=1072.182,316.339,-94.788,174.716,30.425,155.465
C00687=1072.187,316.587,-94.821,174.720,30.430,155.465
C00688=1072.192,316.811,-94.850,174.722,30.434,155.466
C00689=1072.198,317.034,-94.880,174.725,30.439,155.467
C00690=1072.204,317.257,-94.910,174.728,30.442,155.468
C00691=1072.209,317.480,-94.940,174.730,30.447,155.468
C00692=1072.214,317.704,-94.969,174.734,30.451,155.469
C00693=1072.219,317.927,-94.999,174.736,30.455,155.470
C00694=1072.225,318.150,-95.029,174.739,30.459,155.471
C00695=1072.230,318.373,-95.058,174.742,30.463,155.471
C00696=1072.237,318.621,-95.091,174.744,30.468,155.472
C00697=1072.242,318.869,-95.124,174.748,30.472,155.473
C00698=1072.249,319.117,-95.157,174.750,30.477,155.474
C00699=1072.255,319.365,-95.191,174.754,30.482,155.475
C00700=1072.261,319.613,-95.224,174.757,30.486,155.475
C00701=1072.267,319.860,-95.256,174.760,30.491,155.476
C00702=1072.273,320.108,-95.290,174.764,30.496,155.477
C00703=1072.279,320.356,-95.322,174.766,30.501,155.478
C00704=1072.285,320.604,-95.356,174.770,30.505,155.479
C00705=1072.291,320.851,-95.388,174.773,30.509,155.480
C00706=1072.296,321.099,-95.422,174.776,30.514,155.480
C00707=1072.303,321.347,-95.455,174.779,30.519,155.481
C00708=1072.309,321.594,-95.487,174.782,30.524,155.482
C00709=1072.315,321.842,-95.521,174.785,30.528,155.483
C00710=1072.322,322.090,-95.554,174.789,30.533,155.484
C00711=1072.327,322.338,-95.588,174.791,30.537,155.485
C00712=1072.334,322.585,-95.621,174.795,30.542,155.486
C00713=1072.339,322.833,-95.655,174.797,30.547,155.486
C00714=1072.346,323.080,-95.687,174.801,30.552,155.487
C00715=1072.351,323.328,-95.721,174.804,30.556,155.488
C00716=1072.358,323.577,-95.754,174.807,30.561,155.489
C00717=1072.364,323.824,-95.788,174.811,30.566,155.490
C00718=1072.370,324.071,-95.821,174.813,30.571,155.491
C00719=1072.376,324.319,-95.854,174.817,30.575,155.491
C00720=1072.383,324.567,-95.888,174.820,30.580,155.492
C00721=1072.389,324.815,-95.921,174.823,30.584,155.493
C00722=1072.395,325.063,-95.954,174.826,30.589,155.494
C00723=1072.401,325.310,-95.988,174.829,30.594,155.495
C00724=1072.408,325.558,-96.021,174.833,30.599,155.496
C00725=1072.414,325.805,-96.055,174.836,30.603,155.496
C00726=1072.420,326.053,-96.088,174.839,30.608,155.497
C00727=1072.426,326.300,-96.122,174.842,30.613,155.498
C00728=1072.433,326.549,-96.155,174.846,30.617,155.499
C00729=1072.438,326.796,-96.189,174.849,30.622,155.500
C00730=1072.444,327.044,-96.222,174.852,30.627,155.501
C00731=1072.451,327.291,-96.256,174.855,30.632,155.502
C00732=1072.457,327.539,-96.289,174.858,30.636,155.503
C00733=1072.463,327.786,-96.323,174.862,30.641,155.503
C00734=1072.470,328.035,-96.357,174.865,30.646,155.504
C00735=1072.476,328.282,-96.390,174.868,30.650,155.505
C00736=1072.483,328.530,-96.424,174.871,30.655,155.506
C00737=1072.488,328.778,-96.458,174.875,30.660,155.507
C00738=1072.495,329.025,-96.491,174.878,30.665,155.508
C00739=1072.501,329.273,-96.526,174.881,30.670,155.509
C00740=1072.508,329.520,-96.558,174.885,30.675,155.509
C00741=1072.514,329.768,-96.593,174.887,30.679,155.510
C00742=1072.520,330.016,-96.627,174.891,30.684,155.511
C00743=1072.527,330.264,-96.660,174.894,30.689,155.512
C00744=1072.533,330.506,-96.694,174.897,30.693,155.513
C00745=1072.539,330.749,-96.727,174.901,30.698,155.514
C00746=1072.545,330.991,-96.760,174.904,30.702,155.515
C00747=1072.552,331.234,-96.793,174.907,30.707,155.515
C00748=1072.557,331.476,-96.826,174.910,30.712,155.516
C00749=1072.564,331.719,-96.860,174.913,30.717,155.517
C00750=1072.569,331.961,-96.893,174.917,30.722,155.518
C00751=1072.575,332.204,-96.926,174.920,30.727,155.519
C00752=1072.581,332.452,-96.960,174.923,30.732,155.520
C00753=1072.587,332.699,-96.994,174.926,30.736,155.521
C00754=1072.594,332.947,-97.029,174.930,30.741,155.522
C00755=1072.600,333.194,-97.063,174.933,30.746,155.523
C00756=1072.606,333.442,-97.097,174.936,30.751,155.524
C00757=1072.612,333.689,-97.131,174.939,30.756,155.524
C00758=1072.618,333.937,-97.166,174.943,30.761,155.525
C00759=1072.624,334.185,-97.200,174.947,30.766,155.526
C00760=1072.631,334.433,-97.234,174.949,30.771,155.527
C00761=1072.637,334.680,-97.268,174.953,30.777,155.528
C00762=1072.643,334.928,-97.303,174.956,30.782,155.529
C00763=1072.649,335.175,-97.337,174.959,30.786,155.530
C00764=1072.656,335.423,-97.372,174.963,30.791,155.531
C00765=1072.662,335.670,-97.406,174.966,30.796,155.532
C00766=1072.668,335.918,-97.440,174.969,30.801,155.533
C00767=1072.674,336.165,-97.475,174.973,30.806,155.534
C00768=1072.680,336.413,-97.509,174.976,30.811,155.535
C00769=1072.686,336.660,-97.543,174.980,30.816,155.535
C00770=1072.693,336.908,-97.578,174.982,30.821,155.537
C00771=1072.699,337.156,-97.613,174.986,30.826,155.537
C00772=1072.705,337.381,-97.644,174.989,30.831,155.538
C00773=1072.711,337.606,-97.675,174.992,30.836,155.539
C00774=1072.717,337.830,-97.706,174.995,30.840,155.540
C00775=1072.722,338.056,-97.738,174.999,30.845,155.541
C00776=1072.728,338.281,-97.770,175.001,30.849,155.542
C00777=1072.734,338.506,-97.801,175.004,30.854,155.543
C00778=1072.739,338.731,-97.833,175.008,30.858,155.543
C00779=1072.744,338.956,-97.864,175.010,30.863,155.544
C00780=1072.751,339.204,-97.899,175.014,30.868,155.545
C00781=1072.757,339.452,-97.933,175.017,30.874,155.546
C00782=1072.763,339.699,-97.968,175.021,30.879,155.547
C00783=1072.769,339.947,-98.003,175.024,30.884,155.548
C00784=1072.775,340.194,-98.038,175.027,30.889,155.549
C00785=1072.782,340.442,-98.072,175.031,30.894,155.550
C00786=1072.788,340.690,-98.108,175.035,30.899,155.551
C00787=1072.794,340.937,-98.142,175.037,30.904,155.552
C00788=1072.801,341.184,-98.177,175.041,30.910,155.553
C00789=1072.807,341.432,-98.212,175.044,30.915,155.554
C00790=1072.812,341.679,-98.247,175.048,30.920,155.555
C00791=1072.819,341.927,-98.282,175.052,30.925,155.556
C00792=1072.826,342.175,-98.316,175.054,30.930,155.557
C00793=1072.832,342.422,-98.351,175.058,30.935,155.558
C00794=1072.838,342.669,-98.387,175.062,30.941,155.559
C00795=1072.844,342.917,-98.421,175.065,30.946,155.560
C00796=1072.851,343.164,-98.456,175.069,30.951,155.561
C00797=1072.857,343.412,-98.492,175.072,30.956,155.562
C00798=1072.863,343.659,-98.527,175.075,30.962,155.563
C00799=1072.870,343.907,-98.561,175.079,30.967,155.564
C00800=1072.876,344.124,-98.593,175.081,30.971,155.565
C00801=1072.881,344.342,-98.623,175.085,30.976,155.566
C00802=1072.887,344.560,-98.654,175.088,30.980,155.566
C00803=1072.891,344.777,-98.685,175.090,30.985,155.567
C00804=1072.897,344.995,-98.717,175.094,30.990,155.568
C00805=1072.902,345.212,-98.748,175.097,30.995,155.569
C00806=1072.908,345.430,-98.778,175.100,30.999,155.570
C00807=1072.913,345.647,-98.810,175.103,31.004,155.571
C00808=1072.920,345.894,-98.845,175.107,31.010,155.572
C00809=1072.926,346.142,-98.881,175.110,31.015,155.573
C00810=1072.933,346.390,-98.916,175.113,31.020,155.574
C00811=1072.939,346.637,-98.951,175.117,31.025,155.575
C00812=1072.944,346.884,-98.987,175.120,31.031,155.576
C00813=1072.951,347.132,-99.022,175.124,31.036,155.577
C00814=1072.957,347.379,-99.058,175.128,31.042,155.578
C00815=1072.964,347.627,-99.093,175.131,31.047,155.579
C00816=1072.970,347.874,-99.128,175.135,31.053,155.580
C00817=1072.977,348.122,-99.164,175.138,31.058,155.581
C00818=1072.983,348.369,-99.199,175.141,31.063,155.582
C00819=1072.988,348.616,-99.235,175.145,31.069,155.583
C00820=1072.995,348.864,-99.270,175.148,31.074,155.584
C00821=1073.001,349.111,-99.306,175.152,31.080,155.585
C00822=1073.008,349.358,-99.341,175.156,31.085,155.586
C00823=1073.014,349.606,-99.377,175.159,31.091,155.587
C00824=1073.020,349.853,-99.413,175.163,31.096,155.588
C00825=1073.027,350.101,-99.448,175.167,31.102,155.589
C00826=1073.033,350.348,-99.484,175.169,31.107,155.590
C00827=1073.039,350.596,-99.520,175.173,31.112,155.591
C00828=1073.046,350.843,-99.555,175.177,31.118,155.592
C00829=1073.052,351.091,-99.591,175.180,31.123,155.594
C00830=1073.058,351.338,-99.628,175.184,31.129,155.595
C00831=1073.065,351.585,-99.663,175.188,31.134,155.596
C00832=1073.072,351.832,-99.699,175.191,31.140,155.597
C00833=1073.078,352.080,-99.735,175.195,31.146,155.598
C00834=1073.084,352.327,-99.771,175.198,31.151,155.599
C00835=1073.091,352.574,-99.806,175.202,31.156,155.600
C00836=1073.097,352.822,-99.842,175.206,31.162,155.601
C00837=1073.103,353.069,-99.879,175.209,31.168,155.602
C00838=1073.109,353.317,-99.914,175.213,31.173,155.603
C00839=1073.115,353.564,-99.951,175.217,31.179,155.604
C00840=1073.121,353.811,-99.986,175.220,31.185,155.605
C00841=1073.129,354.058,-100.022,175.223,31.190,155.606
C00842=1073.135,354.305,-100.059,175.227,31.196,155.608
C00843=1073.141,354.553,-100.095,175.230,31.201,155.609
C00844=1073.147,354.800,-100.131,175.234,31.207,155.610
C00845=1073.154,355.047,-100.167,175.238,31.213,155.611
C00846=1073.160,355.295,-100.203,175.241,31.219,155.612
C00847=1073.166,355.542,-100.240,175.245,31.224,155.613
C00848=1073.172,355.789,-100.276,175.249,31.230,155.614
C00849=1073.179,356.037,-100.312,175.252,31.236,155.615
C00850=1073.185,356.284,-100.349,175.256,31.242,155.616
C00851=1073.192,356.531,-100.385,175.260,31.247,155.617
C00852=1073.198,356.778,-100.421,175.263,31.253,155.619
C00853=1073.205,357.026,-100.457,175.267,31.259,155.620
C00854=1073.211,357.273,-100.493,175.270,31.264,155.621
C00855=1073.217,357.520,-100.529,175.274,31.270,155.622
C00856=1073.223,357.740,-100.562,175.278,31.275,155.623
C00857=1073.229,357.958,-100.595,175.281,31.280,155.624
C00858=1073.235,358.178,-100.627,175.284,31.286,155.625
C00859=1073.241,358.397,-100.659,175.287,31.291,155.626
C00860=1073.245,358.617,-100.691,175.291,31.296,155.627
C00861=1073.252,358.836,-100.724,175.294,31.301,155.628
C00862=1073.257,359.055,-100.756,175.297,31.306,155.629
C00863=1073.263,359.275,-100.789,175.301,31.312,155.630
C00864=1073.269,359.522,-100.825,175.304,31.318,155.631
C00865=1073.276,359.769,-100.862,175.308,31.323,155.632
C00866=1073.282,360.016,-100.898,175.312,31.329,155.633
C00867=1073.289,360.264,-100.935,175.315,31.335,155.635
C00868=1073.296,360.511,-100.972,175.319,31.341,155.636
C00869=1073.302,360.758,-101.009,175.323,31.347,155.637
C00870=1073.307,361.005,-101.046,175.326,31.353,155.638
C00871=1073.314,361.253,-101.083,175.330,31.359,155.639
C00872=1073.321,361.500,-101.119,175.334,31.364,155.640
C00873=1073.327,361.747,-101.155,175.337,31.370,155.642
C00874=1073.334,361.994,-101.193,175.341,31.376,155.643
C00875=1073.341,362.241,-101.229,175.345,31.382,155.644
C00876=1073.346,362.488,-101.266,175.349,31.388,155.645
C00877=1073.353,362.735,-101.303,175.353,31.395,155.646
C00878=1073.360,362.983,-101.340,175.357,31.401,155.648
C00879=1073.366,363.230,-101.377,175.360,31.407,155.649
C00880=1073.372,363.477,-101.414,175.364,31.413,155.650
C00881=1073.379,363.724,-101.451,175.368,31.418,155.651
C00882=1073.385,363.971,-101.488,175.371,31.425,155.652
C00883=1073.393,364.218,-101.525,175.375,31.431,155.654
C00884=1073.398,364.466,-101.562,175.379,31.437,155.655
C00885=1073.405,364.713,-101.599,175.383,31.443,155.656
C00886=1073.412,364.960,-101.636,175.387,31.449,155.657
C00887=1073.417,365.207,-101.673,175.391,31.455,155.658
C00888=1073.424,365.454,-101.711,175.395,31.462,155.660
C00889=1073.431,365.701,-101.749,175.398,31.468,155.661
C00890=1073.437,365.948,-101.785,175.402,31.474,155.662
C00891=1073.443,366.196,-101.823,175.406,31.480,155.663
C00892=1073.450,366.443,-101.860,175.409,31.486,155.665
C00893=1073.456,366.689,-101.897,175.413,31.492,155.666
C00894=1073.463,366.937,-101.935,175.418,31.499,155.667
C00895=1073.469,367.184,-101.971,175.421,31.505,155.668
C00896=1073.476,367.431,-102.010,175.425,31.511,155.669
C00897=1073.482,367.678,-102.047,175.429,31.518,155.671
C00898=1073.489,367.925,-102.085,175.432,31.523,155.672
C00899=1073.495,368.172,-102.121,175.436,31.530,155.673
C00900=1073.502,368.419,-102.159,175.440,31.536,155.675
C00901=1073.508,368.666,-102.197,175.444,31.543,155.676
C00902=1073.514,368.913,-102.234,175.448,31.549,155.677
C00903=1073.521,369.160,-102.272,175.452,31.555,155.678
C00904=1073.528,369.407,-102.310,175.456,31.562,155.680
C00905=1073.534,369.655,-102.347,175.459,31.568,155.681
C00906=1073.541,369.902,-102.385,175.464,31.575,155.682
C00907=1073.547,370.148,-102.422,175.468,31.581,155.683
C00908=1073.554,370.396,-102.460,175.471,31.587,155.685
C00909=1073.560,370.642,-102.498,175.475,31.593,155.686
C00910=1073.567,370.889,-102.535,175.479,31.600,155.687
C00911=1073.573,371.136,-102.573,175.483,31.606,155.689
C00912=1073.580,371.364,-102.608,175.486,31.612,155.690
C00913=1073.585,371.591,-102.643,175.490,31.618,155.691
C00914=1073.592,371.819,-102.678,175.494,31.624,155.692
C00915=1073.598,372.047,-102.712,175.497,31.630,155.693
C00916=1073.604,372.275,-102.748,175.501,31.636,155.695
C00917=1073.610,372.503,-102.783,175.505,31.642,155.696
C00918=1073.616,372.730,-102.817,175.509,31.648,155.697
C00919=1073.623,372.958,-102.853,175.512,31.654,155.698
C00920=1073.628,373.205,-102.890,175.516,31.661,155.700
C00921=1073.636,373.452,-102.928,175.520,31.667,155.701
C00922=1073.643,373.699,-102.967,175.524,31.674,155.702
C00923=1073.648,373.946,-103.004,175.528,31.680,155.704
C00924=1073.655,374.193,-103.043,175.532,31.687,155.705
C00925=1073.662,374.440,-103.081,175.536,31.693,155.706
C00926=1073.668,374.687,-103.119,175.540,31.700,155.708
C00927=1073.675,374.934,-103.157,175.544,31.707,155.709
C00928=1073.682,375.181,-103.195,175.548,31.714,155.710
C00929=1073.688,375.427,-103.233,175.551,31.720,155.712
C00930=1073.694,375.674,-103.272,175.556,31.727,155.713
C00931=1073.701,375.922,-103.310,175.560,31.734,155.714
C00932=1073.707,376.168,-103.349,175.564,31.740,155.716
C00933=1073.714,376.415,-103.387,175.568,31.747,155.717
C00934=1073.720,376.662,-103.426,175.572,31.754,155.719
C00935=1073.727,376.909,-103.464,175.576,31.761,155.720
C00936=1073.733,377.156,-103.502,175.580,31.768,155.721
C00937=1073.740,377.403,-103.540,175.584,31.774,155.723
C00938=1073.747,377.650,-103.579,175.588,31.781,155.724
C00939=1073.754,377.896,-103.617,175.592,31.788,155.726
C00940=1073.761,378.144,-103.656,175.596,31.795,155.727
C00941=1073.767,378.390,-103.694,175.600,31.802,155.728
C00942=1073.774,378.637,-103.733,175.604,31.808,155.730
C00943=1073.780,378.884,-103.772,175.609,31.815,155.731
C00944=1073.787,379.131,-103.810,175.612,31.822,155.733
C00945=1073.794,379.378,-103.849,175.616,31.829,155.734
C00946=1073.800,379.625,-103.887,175.621,31.836,155.735
C00947=1073.807,379.872,-103.926,175.625,31.843,155.737
C00948=1073.814,380.118,-103.965,175.629,31.850,155.738
C00949=1073.820,380.364,-104.004,175.633,31.857,155.740
C00950=1073.827,380.612,-104.042,175.637,31.864,155.741
C00951=1073.834,380.859,-104.081,175.642,31.871,155.743
C00952=1073.840,381.106,-104.119,175.645,31.878,155.744
C00953=1073.847,381.352,-104.158,175.650,31.885,155.746
C00954=1073.854,381.599,-104.197,175.654,31.892,155.747
C00955=1073.861,381.846,-104.236,175.658,31.899,155.748
C00956=1073.868,382.093,-104.275,175.662,31.906,155.750
C00957=1073.874,382.340,-104.314,175.666,31.913,155.751
C00958=1073.881,382.586,-104.354,175.671,31.920,155.753
C00959=1073.888,382.833,-104.393,175.675,31.928,155.754
C00960=1073.895,383.080,-104.431,175.678,31.934,155.756
C00961=1073.901,383.327,-104.471,175.683,31.942,155.757
C00962=1073.907,383.574,-104.510,175.687,31.949,155.759
C00963=1073.915,383.820,-104.549,175.692,31.956,155.760
C00964=1073.921,384.067,-104.588,175.695,31.964,155.762
C00965=1073.927,384.314,-104.628,175.700,31.971,155.763
C00966=1073.934,384.561,-104.666,175.704,31.978,155.765
C00967=1073.941,384.807,-104.706,175.708,31.985,155.766
C00968=1073.947,385.049,-104.744,175.712,31.992,155.768
C00969=1073.954,385.292,-104.783,175.716,32.000,155.769
C00970=1073.961,385.533,-104.822,175.721,32.007,155.771
C00971=1073.967,385.776,-104.860,175.725,32.014,155.772
C00972=1073.974,386.018,-104.899,175.729,32.022,155.774
C00973=1073.980,386.260,-104.938,175.733,32.029,155.775
C00974=1073.987,386.504,-104.976,175.737,32.036,155.777
C00975=1073.994,386.746,-105.015,175.742,32.043,155.779
C00976=1074.000,386.993,-105.055,175.746,32.051,155.780
C00977=1074.007,387.239,-105.094,175.751,32.058,155.782
C00978=1074.015,387.485,-105.134,175.754,32.066,155.783
C00979=1074.021,387.732,-105.173,175.759,32.073,155.785
C00980=1074.028,387.979,-105.213,175.763,32.080,155.786
C00981=1074.034,388.226,-105.252,175.768,32.088,155.788
C00982=1074.042,388.473,-105.292,175.771,32.095,155.789
C00983=1074.049,388.719,-105.332,175.776,32.103,155.791
C00984=1074.055,388.965,-105.372,175.780,32.111,155.793
C00985=1074.062,389.212,-105.411,175.785,32.118,155.794
C00986=1074.069,389.459,-105.451,175.789,32.125,155.796
C00987=1074.076,389.706,-105.491,175.793,32.133,155.798
C00988=1074.083,389.952,-105.530,175.798,32.141,155.799
C00989=1074.089,390.198,-105.570,175.802,32.148,155.801
C00990=1074.097,390.446,-105.610,175.807,32.156,155.802
C00991=1074.103,390.692,-105.650,175.811,32.164,155.804
C00992=1074.110,390.939,-105.689,175.816,32.172,155.806
C00993=1074.117,391.186,-105.730,175.820,32.179,155.807
C00994=1074.124,391.432,-105.769,175.824,32.187,155.809
C00995=1074.131,391.678,-105.809,175.829,32.195,155.811
C00996=1074.138,391.926,-105.850,175.833,32.203,155.812
C00997=1074.145,392.172,-105.890,175.838,32.210,155.814
C00998=1074.151,392.418,-105.930,175.842,32.218,155.815
C00999=1074.159,392.665,-105.971,175.846,32.226,155.817
C01000=1074.166,392.911,-106.010,175.851,32.234,155.819
C01001=1074.172,393.158,-106.051,175.855,32.242,155.821
C01002=1074.179,393.405,-106.091,175.860,32.250,155.822
C01003=1074.186,393.651,-106.131,175.865,32.258,155.824
C01004=1074.193,393.898,-106.171,175.868,32.266,155.826
C01005=1074.200,394.144,-106.212,175.873,32.274,155.827
C01006=1074.207,394.390,-106.252,175.878,32.281,155.829
C01007=1074.214,394.638,-106.292,175.882,32.289,155.831
C01008=1074.221,394.884,-106.333,175.887,32.298,155.833
C01009=1074.228,395.131,-106.373,175.892,32.306,155.834
C01010=1074.234,395.377,-106.414,175.896,32.314,155.836
C01011=1074.241,395.624,-106.455,175.900,32.322,155.838
C01012=1074.248,395.870,-106.494,175.905,32.330,155.839
C01013=1074.256,396.117,-106.536,175.909,32.338,155.841
C01014=1074.262,396.363,-106.576,175.914,32.346,155.843
C01015=1074.269,396.610,-106.617,175.919,32.355,155.845
C01016=1074.276,396.856,-106.657,175.923,32.362,155.846
C01017=1074.283,397.103,-106.698,175.928,32.371,155.848
C01018=1074.290,397.350,-106.739,175.932,32.379,155.850
C01019=1074.297,397.596,-106.780,175.937,32.387,155.852
C01020=1074.304,397.843,-106.821,175.941,32.396,155.854
C01021=1074.310,398.089,-106.861,175.946,32.404,155.855
C01022=1074.318,398.335,-106.902,175.951,32.413,155.857
C01023=1074.326,398.582,-106.943,175.955,32.420,155.859
C01024=1074.333,398.836,-106.985,175.960,32.429,155.861
C01025=1074.339,399.089,-107.027,175.965,32.438,155.863
C01026=1074.347,399.342,-107.070,175.969,32.447,155.865
C01027=1074.354,399.596,-107.111,175.974,32.455,155.866
C01028=1074.360,399.842,-107.153,175.979,32.464,155.868
C01029=1074.367,400.088,-107.194,175.984,32.472,155.870
C01030=1074.375,400.335,-107.235,175.988,32.481,155.872
C01031=1074.382,400.582,-107.276,175.993,32.489,155.874
C01032=1074.389,400.827,-107.317,175.998,32.498,155.876
C01033=1074.396,401.074,-107.358,176.003,32.507,155.878
C01034=1074.403,401.321,-107.400,176.008,32.515,155.879
C01035=1074.410,401.567,-107.441,176.012,32.524,155.881
C01036=1074.416,401.813,-107.482,176.016,32.532,155.883
C01037=1074.424,402.060,-107.523,176.021,32.541,155.885
C01038=1074.431,402.307,-107.565,176.026,32.549,155.887
C01039=1074.438,402.553,-107.606,176.031,32.558,155.889
C01040=1074.446,402.800,-107.647,176.036,32.567,155.891
C01041=1074.453,403.046,-107.688,176.040,32.576,155.893
C01042=1074.459,403.292,-107.731,176.045,32.585,155.895
C01043=1074.466,403.539,-107.772,176.050,32.593,155.897
C01044=1074.474,403.785,-107.813,176.055,32.602,155.899
C01045=1074.481,404.032,-107.854,176.060,32.611,155.901
C01046=1074.488,404.278,-107.897,176.065,32.620,155.902
C01047=1074.495,404.525,-107.938,176.070,32.629,155.905
C01048=1074.502,404.771,-107.979,176.075,32.638,155.906
C01049=1074.509,405.017,-108.022,176.080,32.647,155.908
C01050=1074.517,405.264,-108.063,176.085,32.656,155.910
C01051=1074.524,405.510,-108.105,176.088,32.665,155.912
C01052=1074.531,405.757,-108.147,176.093,32.674,155.914
C01053=1074.538,406.003,-108.189,176.098,32.683,155.916
C01054=1074.545,406.250,-108.231,176.103,32.692,155.918
C01055=1074.552,406.496,-108.272,176.108,32.701,155.920
C01056=1074.559,406.742,-108.315,176.113,32.710,155.922
C01057=1074.567,406.989,-108.356,176.118,32.719,155.924
C01058=1074.573,407.235,-108.399,176.123,32.728,155.926
C01059=1074.581,407.481,-108.441,176.128,32.738,155.929
C01060=1074.588,407.728,-108.483,176.133,32.747,155.931
C01061=1074.595,407.974,-108.525,176.138,32.756,155.933
C01062=1074.602,408.220,-108.567,176.143,32.766,155.935
C01063=1074.609,408.466,-108.610,176.148,32.775,155.937
C01064=1074.616,408.712,-108.652,176.153,32.785,155.939
C01065=1074.623,408.959,-108.694,176.158,32.794,155.941
C01066=1074.631,409.205,-108.735,176.163,32.803,155.943
C01067=1074.637,409.452,-108.778,176.168,32.813,155.945
C01068=1074.644,409.698,-108.820,176.173,32.822,155.947
C01069=1074.653,409.945,-108.863,176.179,32.831,155.949
C01070=1074.659,410.191,-108.905,176.184,32.841,155.951
C01071=1074.666,410.437,-108.948,176.189,32.851,155.954
C01072=1074.674,410.682,-108.990,176.194,32.860,155.956
C01073=1074.681,410.929,-109.033,176.199,32.869,155.958
C01074=1074.688,411.176,-109.076,176.204,32.879,155.960
C01075=1074.696,411.422,-109.118,176.210,32.889,155.962
C01076=1074.703,411.668,-109.160,176.215,32.898,155.964
C01077=1074.710,411.914,-109.203,176.220,32.908,155.967
C01078=1074.718,412.160,-109.246,176.226,32.918,155.969
C01079=1074.725,412.407,-109.288,176.231,32.928,155.971
C01080=1074.733,412.664,-109.333,176.236,32.937,155.973
C01081=1074.740,412.920,-109.377,176.242,32.948,155.976
C01082=1074.748,413.175,-109.422,176.247,32.958,155.978
C01083=1074.756,413.433,-109.466,176.252,32.968,155.980
C01084=1074.763,413.678,-109.510,176.258,32.978,155.982
C01085=1074.771,413.925,-109.553,176.263,32.988,155.985
C01086=1074.778,414.171,-109.595,176.268,32.998,155.987
C01087=1074.786,414.418,-109.638,176.273,33.008,155.989
C01088=1074.793,414.663,-109.681,176.279,33.018,155.991
C01089=1074.801,414.910,-109.724,176.285,33.028,155.994
C01090=1074.808,415.156,-109.768,176.290,33.038,155.996
C01091=1074.816,415.403,-109.810,176.295,33.048,155.998
C01092=1074.823,415.648,-109.853,176.301,33.058,156.000
C01093=1074.830,415.894,-109.896,176.306,33.068,156.003
C01094=1074.838,416.140,-109.940,176.311,33.079,156.005
C01095=1074.844,416.387,-109.983,176.317,33.089,156.007
C01096=1074.852,416.633,-110.027,176.322,33.099,156.010
C01097=1074.859,416.879,-110.070,176.328,33.109,156.012
C01098=1074.867,417.125,-110.114,176.334,33.120,156.014
C01099=1074.874,417.371,-110.157,176.339,33.130,156.017
C01100=1074.882,417.617,-110.201,176.344,33.140,156.019
C01101=1074.889,417.863,-110.244,176.350,33.151,156.022
C01102=1074.897,418.109,-110.287,176.355,33.161,156.024
C01103=1074.904,418.356,-110.331,176.360,33.172,156.026
C01104=1074.912,418.601,-110.374,176.367,33.182,156.029
C01105=1074.919,418.848,-110.418,176.372,33.193,156.031
C01106=1074.927,419.094,-110.462,176.378,33.203,156.033
C01107=1074.934,419.340,-110.505,176.383,33.214,156.036
C01108=1074.942,419.585,-110.549,176.389,33.224,156.038
C01109=1074.949,419.831,-110.593,176.395,33.235,156.041
C01110=1074.957,420.078,-110.637,176.400,33.245,156.043
C01111=1074.964,420.324,-110.680,176.406,33.256,156.046
C01112=1074.972,420.570,-110.725,176.411,33.267,156.048
C01113=1074.980,420.816,-110.768,176.417,33.278,156.051
C01114=1074.988,421.061,-110.812,176.423,33.289,156.053
C01115=1074.995,421.308,-110.856,176.429,33.300,156.056
C01116=1075.003,421.554,-110.901,176.434,33.310,156.058
C01117=1075.010,421.799,-110.944,176.440,33.321,156.061
C01118=1075.018,422.045,-110.988,176.446,33.332,156.063
C01119=1075.025,422.292,-111.032,176.452,33.343,156.066
C01120=1075.033,422.538,-111.077,176.458,33.354,156.068
C01121=1075.041,422.783,-111.121,176.463,33.365,156.071
C01122=1075.048,423.029,-111.165,176.470,33.376,156.073
C01123=1075.056,423.275,-111.209,176.475,33.388,156.076
C01124=1075.063,423.521,-111.254,176.481,33.398,156.078
C01125=1075.071,423.767,-111.299,176.487,33.410,156.081
C01126=1075.079,424.013,-111.342,176.493,33.421,156.084
C01127=1075.086,424.259,-111.387,176.499,33.432,156.086
C01128=1075.094,424.505,-111.432,176.504,33.444,156.089
C01129=1075.101,424.750,-111.476,176.511,33.455,156.092
C01130=1075.109,424.996,-111.520,176.517,33.466,156.094
C01131=1075.116,425.242,-111.565,176.522,33.477,156.097
C01132=1075.124,425.488,-111.610,176.529,33.489,156.100
C01133=1075.132,425.734,-111.655,176.535,33.501,156.102
C01134=1075.140,425.980,-111.699,176.540,33.512,156.105
C01135=1075.147,426.226,-111.744,176.547,33.523,156.108
C01136=1075.157,426.499,-111.794,176.553,33.536,156.111
C01137=1075.165,426.774,-111.844,176.561,33.549,156.114
C01138=1075.174,427.049,-111.894,176.567,33.562,156.117
C01139=1075.183,427.323,-111.944,176.574,33.575,156.120
C01140=1075.190,427.569,-111.989,176.580,33.587,156.122
C01141=1075.199,427.815,-112.034,176.586,33.599,156.125
C01142=1075.206,428.060,-112.079,176.593,33.610,156.128
C01143=1075.213,428.306,-112.124,176.599,33.622,156.131
C01144=1075.222,428.551,-112.169,176.605,33.634,156.134
C01145=1075.229,428.797,-112.214,176.611,33.646,156.136
C01146=1075.237,429.044,-112.260,176.617,33.658,156.139
C01147=1075.245,429.290,-112.305,176.624,33.670,156.142
C01148=1075.253,429.535,-112.350,176.630,33.682,156.145
C01149=1075.261,429.780,-112.396,176.637,33.694,156.148
C01150=1075.268,430.026,-112.441,176.643,33.706,156.151
C01151=1075.276,430.272,-112.487,176.650,33.718,156.153
C01152=1075.285,430.517,-112.532,176.655,33.730,156.156
C01153=1075.292,430.763,-112.577,176.662,33.743,156.159
C01154=1075.300,431.008,-112.623,176.668,33.755,156.162
C01155=1075.308,431.254,-112.669,176.675,33.767,156.165
C01156=1075.316,431.500,-112.713,176.681,33.779,156.168
C01157=1075.325,431.746,-112.759,176.688,33.792,156.171
C01158=1075.332,431.992,-112.805,176.694,33.804,156.174
C01159=1075.340,432.237,-112.851,176.701,33.816,156.177
C01160=1075.348,432.483,-112.897,176.707,33.829,156.180
C01161=1075.356,432.728,-112.943,176.714,33.842,156.183
C01162=1075.364,432.974,-112.989,176.720,33.854,156.186
C01163=1075.372,433.220,-113.035,176.727,33.867,156.189
C01164=1075.380,433.465,-113.080,176.733,33.880,156.192
C01165=1075.387,433.710,-113.127,176.740,33.892,156.195
C01166=1075.396,433.956,-113.173,176.747,33.905,156.198
C01167=1075.403,434.202,-113.218,176.753,33.918,156.201
C01168=1075.412,434.447,-113.265,176.760,33.931,156.204
C01169=1075.420,434.692,-113.311,176.766,33.944,156.207
C01170=1075.428,434.938,-113.358,176.774,33.957,156.210
C01171=1075.436,435.183,-113.403,176.781,33.969,156.213
C01172=1075.444,435.429,-113.450,176.787,33.983,156.217
C01173=1075.451,435.675,-113.496,176.794,33.995,156.220
C01174=1075.460,435.920,-113.543,176.801,34.008,156.223
C01175=1075.468,436.166,-113.590,176.807,34.022,156.226
C01176=1075.476,436.411,-113.635,176.814,34.035,156.229
C01177=1075.484,436.657,-113.682,176.822,34.048,156.232
C01178=1075.493,436.902,-113.729,176.829,34.061,156.236
C01179=1075.501,437.147,-113.775,176.835,34.074,156.239
C01180=1075.509,437.392,-113.822,176.842,34.088,156.242
C01181=1075.518,437.638,-113.869,176.850,34.101,156.245
C01182=1075.525,437.883,-113.915,176.856,34.115,156.249
C01183=1075.534,438.129,-113.962,176.863,34.128,156.252
C01184=1075.542,438.374,-114.009,176.870,34.142,156.255
C01185=1075.551,438.620,-114.056,176.878,34.155,156.258
C01186=1075.559,438.865,-114.102,176.885,34.168,156.262
C01187=1075.567,439.111,-114.150,176.891,34.182,156.265
C01188=1075.575,439.356,-114.196,176.899,34.196,156.268
C01189=1075.584,439.601,-114.243,176.906,34.210,156.272
C01190=1075.592,439.847,-114.291,176.913,34.223,156.275
C01191=1075.600,440.092,-114.338,176.921,34.238,156.278
C01192=1075.608,440.329,-114.383,176.927,34.251,156.282
C01193=1075.617,440.567,-114.428,176.934,34.264,156.285
C01194=1075.625,440.803,-114.474,176.941,34.278,156.288
C01195=1075.632,441.041,-114.521,176.949,34.291,156.292
C01196=1075.641,441.279,-114.566,176.956,34.305,156.295
C01197=1075.649,441.516,-114.612,176.963,34.319,156.298
C01198=1075.657,441.753,-114.658,176.970,34.333,156.302
C01199=1075.665,441.992,-114.704,176.978,34.346,156.305
C01200=1075.673,442.236,-114.751,176.985,34.360,156.308
C01201=1075.681,442.481,-114.799,176.992,34.375,156.312
C01202=1075.691,442.727,-114.847,176.999,34.389,156.316
C01203=1075.699,442.972,-114.895,177.007,34.403,156.319
C01204=1075.707,443.217,-114.942,177.014,34.418,156.323
C01205=1075.715,443.462,-114.990,177.022,34.433,156.326
C01206=1075.724,443.708,-115.038,177.029,34.447,156.330
C01207=1075.732,443.953,-115.085,177.038,34.462,156.334
C01208=1075.741,444.198,-115.133,177.046,34.476,156.337
C01209=1075.749,444.443,-115.181,177.053,34.491,156.341
C01210=1075.758,444.688,-115.230,177.061,34.506,156.344
C01211=1075.767,444.933,-115.278,177.069,34.521,156.348
C01212=1075.775,445.178,-115.325,177.076,34.535,156.352
C01213=1075.784,445.423,-115.373,177.084,34.550,156.356
C01214=1075.792,445.668,-115.422,177.092,34.565,156.359
C01215=1075.801,445.914,-115.470,177.099,34.580,156.363
C01216=1075.810,446.158,-115.519,177.107,34.595,156.367
C01217=1075.818,446.403,-115.567,177.116,34.611,156.371
C01218=1075.827,446.648,-115.616,177.124,34.626,156.374
C01219=1075.835,446.894,-115.664,177.131,34.641,156.378
C01220=1075.844,447.138,-115.712,177.139,34.656,156.382
C01221=1075.853,447.384,-115.760,177.146,34.671,156.386
C01222=1075.861,447.628,-115.809,177.153,34.687,156.390
C01223=1075.870,447.874,-115.858,177.160,34.702,156.394
C01224=1075.880,448.118,-115.906,177.166,34.717,156.397
C01225=1075.888,448.363,-115.955,177.172,34.732,156.401
C01226=1075.896,448.607,-116.004,177.178,34.747,156.405
C01227=1075.906,448.851,-116.052,177.184,34.762,156.409
C01228=1075.917,449.096,-116.099,177.189,34.777,156.413
C01229=1075.928,449.341,-116.146,177.194,34.790,156.416
C01230=1075.941,449.586,-116.192,177.200,34.804,156.419
C01231=1075.957,449.832,-116.238,177.205,34.816,156.423
C01232=1075.599,449.828,-116.473,177.186,34.971,156.464
C01233=1075.584,449.583,-116.429,177.180,34.958,156.460
C01234=1075.570,449.337,-116.382,177.174,34.945,156.457
C01235=1075.558,449.092,-116.336,177.169,34.931,156.453
C01236=1075.548,448.848,-116.288,177.163,34.917,156.450
C01237=1075.538,448.603,-116.240,177.157,34.902,156.446
C01238=1075.530,448.359,-116.191,177.152,34.887,156.442
C01239=1075.520,448.114,-116.143,177.145,34.872,156.438
C01240=1075.512,447.870,-116.094,177.138,34.856,156.434
C01241=1075.502,447.625,-116.046,177.132,34.842,156.431
C01242=1075.494,447.380,-115.997,177.124,34.826,156.427
C01243=1075.485,447.135,-115.948,177.117,34.811,156.423
C01244=1075.477,446.890,-115.900,177.110,34.796,156.419
C01245=1075.468,446.645,-115.851,177.101,34.781,156.415
C01246=1075.459,446.400,-115.802,177.093,34.765,156.411
C01247=1075.450,446.155,-115.754,177.085,34.750,156.408
C01248=1075.442,445.910,-115.706,177.078,34.735,156.404
C01249=1075.433,445.664,-115.657,177.069,34.720,156.400
C01250=1075.424,445.420,-115.609,177.061,34.705,156.396
C01251=1075.416,445.175,-115.561,177.054,34.690,156.393
C01252=1075.408,444.930,-115.513,177.046,34.675,156.389
C01253=1075.398,444.685,-115.465,177.038,34.661,156.385
C01254=1075.390,444.440,-115.416,177.030,34.646,156.382
C01255=1075.382,444.194,-115.368,177.022,34.631,156.378
C01256=1075.373,443.950,-115.321,177.014,34.617,156.374
C01257=1075.364,443.704,-115.273,177.007,34.602,156.371
C01258=1075.355,443.459,-115.225,176.999,34.588,156.367
C01259=1075.347,443.214,-115.177,176.992,34.573,156.364
C01260=1075.339,442.968,-115.129,176.984,34.559,156.360
C01261=1075.330,442.723,-115.082,176.976,34.544,156.356
C01262=1075.322,442.478,-115.034,176.969,34.530,156.353
C01263=1075.313,442.233,-114.986,176.960,34.515,156.349
C01264=1075.305,441.988,-114.938,176.953,34.501,156.346
C01265=1075.297,441.759,-114.895,176.946,34.488,156.342
C01266=1075.289,441.530,-114.850,176.940,34.475,156.339
C01267=1075.282,441.302,-114.805,176.933,34.462,156.336
C01268=1075.274,441.073,-114.761,176.926,34.449,156.333
C01269=1075.266,440.845,-114.717,176.919,34.436,156.330
C01270=1075.258,440.616,-114.673,176.912,34.423,156.326
C01271=1075.250,440.388,-114.629,176.905,34.410,156.323
C01272=1075.242,440.159,-114.585,176.898,34.397,156.320
C01273=1075.234,439.914,-114.538,176.890,34.383,156.317
C01274=1075.226,439.668,-114.490,176.883,34.369,156.313
C01275=1075.217,439.423,-114.444,176.876,34.355,156.310
C01276=1075.210,439.178,-114.396,176.868,34.342,156.306
C01277=1075.201,438.933,-114.349,176.862,34.328,156.303
C01278=1075.193,438.687,-114.303,176.855,34.314,156.300
C01279=1075.184,438.442,-114.256,176.847,34.301,156.296
C01280=1075.176,438.196,-114.209,176.840,34.287,156.293
C01281=1075.168,437.950,-114.162,176.833,34.274,156.290
C01282=1075.159,437.705,-114.115,176.826,34.260,156.287
C01283=1075.151,437.460,-114.069,176.818,34.247,156.283
C01284=1075.143,437.215,-114.022,176.812,34.233,156.280
C01285=1075.134,436.969,-113.975,176.805,34.220,156.277
C01286=1075.126,436.723,-113.929,176.798,34.207,156.274
C01287=1075.118,436.479,-113.882,176.790,34.194,156.271
C01288=1075.109,436.233,-113.835,176.783,34.181,156.267
C01289=1075.101,435.987,-113.788,176.777,34.168,156.264
C01290=1075.094,435.742,-113.742,176.770,34.155,156.261
C01291=1075.085,435.496,-113.696,176.763,34.141,156.258
C01292=1075.077,435.252,-113.649,176.756,34.129,156.255
C01293=1075.069,435.005,-113.603,176.749,34.116,156.252
C01294=1075.061,434.761,-113.557,176.742,34.103,156.249
C01295=1075.053,434.515,-113.511,176.735,34.090,156.245
C01296=1075.045,434.270,-113.465,176.729,34.077,156.242
C01297=1075.037,434.024,-113.419,176.722,34.064,156.239
C01298=1075.029,433.779,-113.372,176.715,34.052,156.236
C01299=1075.020,433.533,-113.326,176.709,34.039,156.233
C01300=1075.013,433.287,-113.281,176.702,34.026,156.230
C01301=1075.004,433.042,-113.234,176.695,34.014,156.227
C01302=1074.997,432.796,-113.188,176.689,34.001,156.224
C01303=1074.988,432.550,-113.142,176.682,33.988,156.221
C01304=1074.981,432.305,-113.097,176.675,33.975,156.218
C01305=1074.973,432.059,-113.051,176.669,33.963,156.215
C01306=1074.965,431.814,-113.004,176.662,33.950,156.212
C01307=1074.957,431.568,-112.959,176.656,33.938,156.209
C01308=1074.949,431.322,-112.912,176.649,33.926,156.206
C01309=1074.941,431.076,-112.868,176.642,33.914,156.203
C01310=1074.933,430.831,-112.823,176.636,33.902,156.200
C01311=1074.925,430.585,-112.777,176.629,33.889,156.197
C01312=1074.917,430.339,-112.731,176.623,33.877,156.194
C01313=1074.909,430.094,-112.685,176.617,33.865,156.192
C01314=1074.901,429.849,-112.640,176.611,33.853,156.189
C01315=1074.893,429.603,-112.594,176.604,33.841,156.186
C01316=1074.885,429.357,-112.549,176.598,33.829,156.183
C01317=1074.878,429.111,-112.504,176.591,33.817,156.180
C01318=1074.869,428.866,-112.459,176.585,33.805,156.177
C01319=1074.862,428.620,-112.414,176.578,33.793,156.175
C01320=1074.854,428.374,-112.368,176.573,33.781,156.172
C01321=1074.847,428.128,-112.323,176.566,33.770,156.169
C01322=1074.838,427.883,-112.278,176.560,33.757,156.166
C01323=1074.831,427.637,-112.233,176.553,33.745,156.163
C01324=1074.822,427.392,-112.188,176.547,33.734,156.161
C01325=1074.814,427.115,-112.137,176.540,33.721,156.158
C01326=1074.805,426.839,-112.086,176.534,33.708,156.154
C01327=1074.796,426.563,-112.037,176.526,33.695,156.151
C01328=1074.788,426.287,-111.986,176.520,33.682,156.148
C01329=1074.780,426.041,-111.941,176.513,33.671,156.146
C01330=1074.772,425.795,-111.897,176.507,33.659,156.143
C01331=1074.764,425.550,-111.852,176.501,33.648,156.140
C01332=1074.757,425.304,-111.807,176.495,33.636,156.138
C01333=1074.748,425.058,-111.762,176.489,33.625,156.135
C01334=1074.740,424.813,-111.718,176.483,33.613,156.132
C01335=1074.733,424.567,-111.673,176.477,33.602,156.130
C01336=1074.725,424.321,-111.629,176.470,33.591,156.127
C01337=1074.718,424.075,-111.584,176.465,33.580,156.124
C01338=1074.710,423.829,-111.539,176.459,33.569,156.122
C01339=1074.703,423.582,-111.495,176.452,33.557,156.119
C01340=1074.695,423.337,-111.451,176.447,33.546,156.117
C01341=1074.687,423.092,-111.407,176.441,33.535,156.114
C01342=1074.680,422.846,-111.362,176.435,33.524,156.111
C01343=1074.672,422.600,-111.318,176.429,33.513,156.109
C01344=1074.665,422.353,-111.273,176.424,33.502,156.106
C01345=1074.657,422.107,-111.229,176.417,33.490,156.104
C01346=1074.649,421.862,-111.185,176.412,33.480,156.101
C01347=1074.642,421.616,-111.141,176.406,33.469,156.099
C01348=1074.634,421.370,-111.096,176.400,33.458,156.096
C01349=1074.626,421.124,-111.053,176.394,33.447,156.094
C01350=1074.618,420.878,-111.009,176.389,33.436,156.091
C01351=1074.611,420.632,-110.965,176.382,33.426,156.089
C01352=1074.604,420.386,-110.920,176.377,33.415,156.086
C01353=1074.596,420.140,-110.877,176.371,33.404,156.084
C01354=1074.588,419.893,-110.833,176.366,33.394,156.081
C01355=1074.581,419.648,-110.789,176.359,33.383,156.079
C01356=1074.573,419.402,-110.746,176.354,33.373,156.076
C01357=1074.565,419.156,-110.702,176.348,33.362,156.074
C01358=1074.558,418.910,-110.659,176.343,33.351,156.072
C01359=1074.550,418.664,-110.615,176.337,33.341,156.069
C01360=1074.542,418.418,-110.571,176.331,33.330,156.067
C01361=1074.536,418.172,-110.527,176.326,33.320,156.064
C01362=1074.528,417.925,-110.483,176.320,33.309,156.062
C01363=1074.520,417.679,-110.440,176.314,33.299,156.060
C01364=1074.513,417.433,-110.396,176.309,33.289,156.057
C01365=1074.505,417.187,-110.353,176.303,33.278,156.055
C01366=1074.498,416.941,-110.309,176.298,33.268,156.052
C01367=1074.490,416.695,-110.266,176.293,33.258,156.050
C01368=1074.483,416.449,-110.223,176.286,33.247,156.048
C01369=1074.476,416.202,-110.180,176.281,33.237,156.045
C01370=1074.469,415.957,-110.136,176.276,33.227,156.043
C01371=1074.461,415.710,-110.093,176.270,33.217,156.041
C01372=1074.454,415.465,-110.050,176.265,33.206,156.038
C01373=1074.446,415.218,-110.006,176.259,33.196,156.036
C01374=1074.439,414.972,-109.963,176.254,33.187,156.034
C01375=1074.431,414.726,-109.920,176.248,33.176,156.032
C01376=1074.424,414.480,-109.878,176.243,33.166,156.029
C01377=1074.416,414.233,-109.834,176.238,33.157,156.027
C01378=1074.409,413.988,-109.791,176.233,33.147,156.025
C01379=1074.401,413.741,-109.748,176.227,33.137,156.023
C01380=1074.393,413.495,-109.705,176.221,33.127,156.020
C01381=1074.386,413.237,-109.660,176.216,33.117,156.018
C01382=1074.378,412.979,-109.615,176.210,33.106,156.016
C01383=1074.371,412.721,-109.571,176.205,33.096,156.013
C01384=1074.363,412.463,-109.526,176.199,33.086,156.011
C01385=1074.356,412.217,-109.483,176.194,33.076,156.009
C01386=1074.347,411.971,-109.440,176.189,33.066,156.007
C01387=1074.340,411.724,-109.398,176.184,33.057,156.005
C01388=1074.334,411.478,-109.355,176.178,33.047,156.002
C01389=1074.327,411.232,-109.313,176.173,33.037,156.000
C01390=1074.318,410.986,-109.270,176.168,33.028,155.998
C01391=1074.311,410.739,-109.227,176.163,33.018,155.996
C01392=1074.304,410.493,-109.185,176.157,33.009,155.994
C01393=1074.297,410.247,-109.143,176.152,32.999,155.992
C01394=1074.289,410.000,-109.100,176.147,32.989,155.989
C01395=1074.282,409.754,-109.058,176.142,32.980,155.987
C01396=1074.275,409.508,-109.015,176.137,32.971,155.985
C01397=1074.268,409.262,-108.973,176.132,32.961,155.983
C01398=1074.261,409.016,-108.931,176.127,32.952,155.981
C01399=1074.254,408.769,-108.888,176.122,32.943,155.979
C01400=1074.246,408.522,-108.845,176.116,32.933,155.977
C01401=1074.239,408.276,-108.803,176.111,32.924,155.975
C01402=1074.232,408.030,-108.761,176.106,32.915,155.973
C01403=1074.224,407.784,-108.719,176.101,32.905,155.971
C01404=1074.218,407.537,-108.677,176.096,32.896,155.968
C01405=1074.211,407.291,-108.635,176.091,32.887,155.967
C01406=1074.203,407.045,-108.593,176.086,32.878,155.964
C01407=1074.196,406.799,-108.550,176.081,32.868,155.962
C01408=1074.189,406.552,-108.509,176.076,32.859,155.960
C01409=1074.182,406.306,-108.466,176.071,32.850,155.958
C01410=1074.175,406.059,-108.425,176.066,32.841,155.956
C01411=1074.167,405.813,-108.383,176.061,32.832,155.954
C01412=1074.160,405.567,-108.341,176.056,32.823,155.952
C01413=1074.153,405.320,-108.299,176.051,32.814,155.950
C01414=1074.146,405.074,-108.257,176.046,32.805,155.948
C01415=1074.139,404.827,-108.216,176.042,32.796,155.946
C01416=1074.131,404.581,-108.174,176.037,32.787,155.944
C01417=1074.125,404.335,-108.132,176.032,32.778,155.942
C01418=1074.118,404.088,-108.091,176.027,32.769,155.940
C01419=1074.110,403.842,-108.049,176.022,32.760,155.938
C01420=1074.103,403.595,-108.007,176.017,32.751,155.936
C01421=1074.096,403.348,-107.966,176.012,32.742,155.935
C01422=1074.089,403.103,-107.924,176.007,32.734,155.933
C01423=1074.082,402.857,-107.883,176.003,32.725,155.931
C01424=1074.075,402.610,-107.842,175.998,32.716,155.929
C01425=1074.068,402.363,-107.800,175.993,32.708,155.927
C01426=1074.061,402.117,-107.759,175.988,32.699,155.925
C01427=1074.053,401.870,-107.717,175.983,32.690,155.923
C01428=1074.046,401.624,-107.675,175.978,32.682,155.921
C01429=1074.039,401.378,-107.635,175.974,32.673,155.919
C01430=1074.032,401.131,-107.593,175.969,32.664,155.917
C01431=1074.025,400.885,-107.551,175.964,32.656,155.916
C01432=1074.018,400.638,-107.510,175.959,32.647,155.914
C01433=1074.011,400.391,-107.469,175.954,32.639,155.912
C01434=1074.004,400.145,-107.428,175.950,32.630,155.910
C01435=1073.997,399.899,-107.387,175.945,32.622,155.908
C01436=1073.990,399.652,-107.346,175.941,32.613,155.906
C01437=1073.982,399.397,-107.304,175.936,32.605,155.904
C01438=1073.976,399.143,-107.261,175.931,32.596,155.902
C01439=1073.968,398.888,-107.219,175.926,32.587,155.901
C01440=1073.961,398.633,-107.177,175.921,32.578,155.899
C01441=1073.954,398.387,-107.136,175.917,32.570,155.897
C01442=1073.947,398.140,-107.095,175.912,32.562,155.895
C01443=1073.940,397.893,-107.054,175.907,32.553,155.893
C01444=1073.933,397.647,-107.013,175.903,32.545,155.891
C01445=1073.926,397.401,-106.972,175.898,32.537,155.890
C01446=1073.919,397.154,-106.932,175.893,32.529,155.888
C01447=1073.912,396.907,-106.891,175.888,32.521,155.886
C01448=1073.905,396.661,-106.849,175.884,32.512,155.884
C01449=1073.898,396.414,-106.809,175.880,32.504,155.882
C01450=1073.891,396.168,-106.768,175.875,32.496,155.881
C01451=1073.884,395.922,-106.728,175.871,32.488,155.879
C01452=1073.877,395.675,-106.687,175.866,32.480,155.877
C01453=1073.870,395.428,-106.647,175.861,32.472,155.876
C01454=1073.863,395.182,-106.606,175.857,32.463,155.874
C01455=1073.857,394.935,-106.566,175.852,32.455,155.872
C01456=1073.850,394.688,-106.525,175.847,32.448,155.870
C01457=1073.843,394.442,-106.484,175.843,32.439,155.869
C01458=1073.835,394.195,-106.444,175.838,32.431,155.867
C01459=1073.829,393.949,-106.404,175.834,32.423,155.865
C01460=1073.821,393.702,-106.363,175.830,32.415,155.863
C01461=1073.815,393.456,-106.323,175.825,32.408,155.862
C01462=1073.808,393.209,-106.283,175.821,32.400,155.860
C01463=1073.801,392.962,-106.243,175.816,32.392,155.858
C01464=1073.795,392.716,-106.203,175.811,32.384,155.857
C01465=1073.787,392.469,-106.162,175.807,32.376,155.855
C01466=1073.780,392.223,-106.122,175.802,32.368,155.853
C01467=1073.774,391.976,-106.082,175.799,32.360,155.852
C01468=1073.766,391.730,-106.042,175.794,32.353,155.850
C01469=1073.760,391.483,-106.002,175.789,32.345,155.848
C01470=1073.753,391.236,-105.962,175.785,32.337,155.847
C01471=1073.746,390.990,-105.922,175.780,32.329,155.845
C01472=1073.738,390.743,-105.882,175.776,32.322,155.843
C01473=1073.732,390.497,-105.842,175.771,32.314,155.842
C01474=1073.724,390.250,-105.802,175.767,32.306,155.840
C01475=1073.718,390.003,-105.762,175.763,32.298,155.838
C01476=1073.711,389.757,-105.722,175.758,32.291,155.837
C01477=1073.705,389.510,-105.683,175.754,32.284,155.835
C01478=1073.697,389.263,-105.643,175.749,32.276,155.834
C01479=1073.690,389.017,-105.603,175.745,32.268,155.832
C01480=1073.684,388.770,-105.563,175.740,32.261,155.830
C01481=1073.676,388.524,-105.524,175.737,32.253,155.829
C01482=1073.670,388.276,-105.484,175.732,32.245,155.827
C01483=1073.663,388.030,-105.444,175.727,32.238,155.826
C01484=1073.656,387.784,-105.405,175.723,32.231,155.824
C01485=1073.649,387.537,-105.365,175.718,32.223,155.823
C01486=1073.642,387.291,-105.326,175.714,32.216,155.821
C01487=1073.635,387.043,-105.285,175.710,32.208,155.819
C01488=1073.629,386.797,-105.246,175.706,32.201,155.818
C01489=1073.622,386.554,-105.208,175.702,32.194,155.816
C01490=1073.616,386.311,-105.169,175.697,32.186,155.815
C01491=1073.609,386.067,-105.130,175.693,32.179,155.813
C01492=1073.602,385.824,-105.091,175.688,32.172,155.812
C01493=1073.596,385.582,-105.052,175.685,32.164,155.810
C01494=1073.588,385.339,-105.014,175.681,32.158,155.809
C01495=1073.582,385.096,-104.975,175.676,32.150,155.807
C01496=1073.575,384.853,-104.936,175.672,32.143,155.806
C01497=1073.568,384.606,-104.897,175.667,32.136,155.804
C01498=1073.562,384.359,-104.857,175.664,32.128,155.803
C01499=1073.555,384.112,-104.818,175.659,32.121,155.801
C01500=1073.548,383.866,-104.779,175.655,32.114,155.800
C01501=1073.542,383.618,-104.740,175.651,32.107,155.798
C01502=1073.535,383.372,-104.700,175.646,32.099,155.796
C01503=1073.528,383.125,-104.661,175.643,32.092,155.795
C01504=1073.522,382.879,-104.623,175.638,32.085,155.793
C01505=1073.516,382.632,-104.583,175.634,32.078,155.792
C01506=1073.509,382.385,-104.544,175.630,32.071,155.790
C01507=1073.502,382.139,-104.505,175.625,32.064,155.789
C01508=1073.496,381.892,-104.465,175.622,32.056,155.787
C01509=1073.489,381.645,-104.427,175.617,32.049,155.786
C01510=1073.482,381.398,-104.388,175.613,32.042,155.785
C01511=1073.475,381.151,-104.349,175.609,32.035,155.783
C01512=1073.468,380.905,-104.310,175.604,32.028,155.782
C01513=1073.462,380.658,-104.271,175.601,32.021,155.780
C01514=1073.455,380.411,-104.232,175.596,32.014,155.779
C01515=1073.448,380.164,-104.194,175.592,32.007,155.777
C01516=1073.441,379.917,-104.155,175.588,32.000,155.776
C01517=1073.435,379.670,-104.117,175.583,31.993,155.774
C01518=1073.428,379.423,-104.078,175.580,31.986,155.773
C01519=1073.421,379.176,-104.039,175.576,31.980,155.772
C01520=1073.415,378.930,-104.000,175.571,31.973,155.770
C01521=1073.408,378.683,-103.962,175.567,31.966,155.769
C01522=1073.402,378.436,-103.923,175.564,31.959,155.767
C01523=1073.394,378.189,-103.885,175.559,31.952,155.766
C01524=1073.387,377.943,-103.846,175.555,31.945,155.765
C01525=1073.381,377.695,-103.808,175.551,31.939,155.763
C01526=1073.374,377.448,-103.769,175.546,31.932,155.762
C01527=1073.368,377.202,-103.731,175.543,31.925,155.760
C01528=1073.361,376.955,-103.693,175.539,31.918,155.759
C01529=1073.354,376.708,-103.654,175.535,31.911,155.758
C01530=1073.347,376.461,-103.615,175.530,31.904,155.756
C01531=1073.342,376.214,-103.577,175.527,31.898,155.755
C01532=1073.335,375.967,-103.539,175.523,31.891,155.753
C01533=1073.328,375.720,-103.500,175.518,31.884,155.752
C01534=1073.321,375.473,-103.462,175.514,31.878,155.751
C01535=1073.315,375.227,-103.424,175.511,31.871,155.749
C01536=1073.308,374.980,-103.386,175.507,31.864,155.748
C01537=1073.301,374.732,-103.348,175.502,31.857,155.746
C01538=1073.296,374.486,-103.310,175.498,31.851,155.745
C01539=1073.289,374.239,-103.271,175.495,31.844,155.744
C01540=1073.282,373.991,-103.233,175.491,31.838,155.742
C01541=1073.276,373.745,-103.194,175.486,31.831,155.741
C01542=1073.269,373.498,-103.157,175.482,31.824,155.740
C01543=1073.262,373.251,-103.119,175.479,31.818,155.738
C01544=1073.256,373.004,-103.081,175.475,31.811,155.737
C01545=1073.249,372.775,-103.046,175.471,31.805,155.736
C01546=1073.244,372.547,-103.010,175.467,31.799,155.735
C01547=1073.237,372.318,-102.976,175.464,31.793,155.733
C01548=1073.232,372.090,-102.940,175.460,31.788,155.732
C01549=1073.225,371.862,-102.905,175.456,31.781,155.731
C01550=1073.219,371.634,-102.871,175.452,31.775,155.730
C01551=1073.213,371.405,-102.835,175.448,31.769,155.729
C01552=1073.207,371.177,-102.801,175.445,31.764,155.727
C01553=1073.200,370.929,-102.763,175.441,31.757,155.726
C01554=1073.194,370.683,-102.726,175.437,31.751,155.725
C01555=1073.187,370.435,-102.687,175.433,31.744,155.724
C01556=1073.181,370.189,-102.650,175.430,31.738,155.722
C01557=1073.174,369.941,-102.612,175.425,31.731,155.721
C01558=1073.168,369.694,-102.574,175.421,31.725,155.720
C01559=1073.161,369.448,-102.537,175.418,31.719,155.718
C01560=1073.154,369.200,-102.499,175.414,31.713,155.717
C01561=1073.148,368.954,-102.462,175.410,31.706,155.716
C01562=1073.141,368.706,-102.423,175.406,31.700,155.715
C01563=1073.135,368.460,-102.386,175.402,31.693,155.713
C01564=1073.128,368.212,-102.348,175.398,31.687,155.712
C01565=1073.121,367.966,-102.311,175.394,31.681,155.711
C01566=1073.115,367.718,-102.274,175.390,31.675,155.709
C01567=1073.109,367.471,-102.236,175.387,31.668,155.708
C01568=1073.102,367.224,-102.198,175.383,31.662,155.707
C01569=1073.095,366.978,-102.161,175.379,31.656,155.706
C01570=1073.090,366.730,-102.124,175.375,31.649,155.704
C01571=1073.083,366.483,-102.087,175.371,31.643,155.703
C01572=1073.077,366.236,-102.049,175.367,31.637,155.702
C01573=1073.070,365.989,-102.012,175.363,31.631,155.701
C01574=1073.064,365.742,-101.974,175.360,31.625,155.699
C01575=1073.057,365.494,-101.937,175.356,31.619,155.698
C01576=1073.051,365.247,-101.900,175.352,31.612,155.697
C01577=1073.044,365.001,-101.863,175.349,31.606,155.696
C01578=1073.037,364.753,-101.826,175.345,31.600,155.695
C01579=1073.032,364.506,-101.788,175.340,31.594,155.693
C01580=1073.025,364.259,-101.752,175.336,31.588,155.692
C01581=1073.018,364.012,-101.715,175.333,31.582,155.691
C01582=1073.012,363.765,-101.678,175.329,31.576,155.690
C01583=1073.005,363.517,-101.640,175.325,31.570,155.689
C01584=1072.999,363.271,-101.603,175.322,31.564,155.687
C01585=1072.992,363.024,-101.567,175.318,31.557,155.686
C01586=1072.986,362.776,-101.530,175.314,31.551,155.685
C01587=1072.980,362.529,-101.492,175.310,31.546,155.684
C01588=1072.973,362.282,-101.456,175.307,31.540,155.683
C01589=1072.966,362.034,-101.419,175.303,31.534,155.681
C01590=1072.960,361.788,-101.382,175.299,31.528,155.680
C01591=1072.953,361.541,-101.345,175.296,31.522,155.679
C01592=1072.947,361.293,-101.308,175.292,31.516,155.678
C01593=1072.941,361.046,-101.271,175.287,31.510,155.677
C01594=1072.935,360.799,-101.235,175.283,31.504,155.676
C01595=1072.928,360.552,-101.198,175.280,31.498,155.674
C01596=1072.921,360.304,-101.161,175.276,31.492,155.673
C01597=1072.915,360.057,-101.124,175.272,31.486,155.672
C01598=1072.908,359.810,-101.088,175.269,31.480,155.671
C01599=1072.903,359.563,-101.051,175.265,31.474,155.670
C01600=1072.896,359.315,-101.014,175.261,31.468,155.669
C01601=1072.890,359.095,-100.982,175.259,31.463,155.667
C01602=1072.884,358.875,-100.949,175.255,31.458,155.667
C01603=1072.878,358.655,-100.917,175.252,31.453,155.665
C01604=1072.873,358.436,-100.884,175.248,31.448,155.664
C01605=1072.868,358.216,-100.852,175.245,31.443,155.663
C01606=1072.861,357.996,-100.819,175.242,31.438,155.662
C01607=1072.856,357.776,-100.787,175.238,31.432,155.661
C01608=1072.850,357.556,-100.754,175.235,31.427,155.660
C01609=1072.844,357.308,-100.719,175.232,31.421,155.659
C01610=1072.837,357.060,-100.682,175.228,31.416,155.658
C01611=1072.830,356.813,-100.645,175.224,31.410,155.657
C01612=1072.824,356.566,-100.609,175.221,31.404,155.656
C01613=1072.818,356.319,-100.572,175.217,31.399,155.655
C01614=1072.811,356.072,-100.536,175.213,31.393,155.654
C01615=1072.805,355.825,-100.500,175.210,31.387,155.653
C01616=1072.799,355.578,-100.464,175.206,31.381,155.651
C01617=1072.792,355.330,-100.427,175.202,31.375,155.650
C01618=1072.786,355.083,-100.391,175.199,31.370,155.649
C01619=1072.779,354.835,-100.355,175.195,31.364,155.648
C01620=1072.773,354.588,-100.319,175.191,31.359,155.647
C01621=1072.766,354.341,-100.283,175.188,31.353,155.646
C01622=1072.760,354.094,-100.247,175.184,31.347,155.645
C01623=1072.754,353.846,-100.210,175.180,31.341,155.644
C01624=1072.748,353.599,-100.175,175.176,31.336,155.643
C01625=1072.742,353.352,-100.138,175.173,31.330,155.642
C01626=1072.736,353.104,-100.102,175.169,31.325,155.640
C01627=1072.729,352.857,-100.067,175.165,31.319,155.639
C01628=1072.722,352.610,-100.031,175.163,31.313,155.638
C01629=1072.716,352.363,-99.994,175.159,31.308,155.637
C01630=1072.710,352.115,-99.959,175.155,31.302,155.636
C01631=1072.704,351.868,-99.922,175.152,31.297,155.635
C01632=1072.697,351.621,-99.887,175.148,31.291,155.634
C01633=1072.691,351.373,-99.851,175.144,31.286,155.633
C01634=1072.685,351.126,-99.815,175.141,31.280,155.632
C01635=1072.678,350.878,-99.780,175.137,31.275,155.631
C01636=1072.672,350.631,-99.743,175.133,31.269,155.630
C01637=1072.666,350.384,-99.708,175.130,31.264,155.629
C01638=1072.659,350.136,-99.673,175.127,31.259,155.628
C01639=1072.652,349.889,-99.636,175.123,31.253,155.627
C01640=1072.646,349.642,-99.600,175.120,31.247,155.625
C01641=1072.640,349.394,-99.565,175.116,31.242,155.624
C01642=1072.634,349.147,-99.530,175.112,31.236,155.623
C01643=1072.628,348.899,-99.494,175.109,31.231,155.622
C01644=1072.620,348.652,-99.458,175.105,31.225,155.621
C01645=1072.614,348.404,-99.422,175.101,31.220,155.620
C01646=1072.608,348.157,-99.387,175.099,31.215,155.619
C01647=1072.602,347.910,-99.352,175.095,31.209,155.618
C01648=1072.596,347.662,-99.316,175.091,31.204,155.617
C01649=1072.589,347.415,-99.281,175.088,31.198,155.616
C01650=1072.583,347.167,-99.245,175.084,31.193,155.615
C01651=1072.577,346.920,-99.210,175.080,31.188,155.614
C01652=1072.571,346.672,-99.174,175.077,31.182,155.613
C01653=1072.564,346.425,-99.139,175.074,31.177,155.612
C01654=1072.558,346.177,-99.103,175.070,31.172,155.611
C01655=1072.552,345.931,-99.069,175.067,31.166,155.610
C01656=1072.546,345.683,-99.033,175.063,31.161,155.609
C01657=1072.540,345.465,-99.002,175.060,31.156,155.608
C01658=1072.535,345.246,-98.971,175.057,31.152,155.607
C01659=1072.529,345.028,-98.940,175.054,31.147,155.606
C01660=1072.523,344.810,-98.909,175.051,31.142,155.605
C01661=1072.518,344.592,-98.877,175.047,31.138,155.605
C01662=1072.513,344.374,-98.846,175.045,31.133,155.604
C01663=1072.506,344.155,-98.815,175.042,31.128,155.603
C01664=1072.501,343.936,-98.784,175.038,31.124,155.602
C01665=1072.495,343.690,-98.749,175.035,31.118,155.601
C01666=1072.488,343.442,-98.714,175.032,31.113,155.600
C01667=1072.482,343.195,-98.679,175.028,31.108,155.599
C01668=1072.476,342.947,-98.644,175.025,31.102,155.598
C01669=1072.469,342.699,-98.608,175.021,31.097,155.597
C01670=1072.463,342.453,-98.574,175.017,31.092,155.596
C01671=1072.457,342.204,-98.539,175.015,31.087,155.595
C01672=1072.451,341.957,-98.504,175.011,31.082,155.594
C01673=1072.444,341.710,-98.469,175.007,31.076,155.593
C01674=1072.439,341.462,-98.434,175.004,31.071,155.592
C01675=1072.432,341.215,-98.399,175.001,31.066,155.591
C01676=1072.425,340.967,-98.364,174.997,31.061,155.590
C01677=1072.419,340.720,-98.329,174.994,31.056,155.589
C01678=1072.413,340.472,-98.294,174.990,31.051,155.588
C01679=1072.407,340.224,-98.259,174.987,31.046,155.587
C01680=1072.401,339.978,-98.225,174.984,31.040,155.586
C01681=1072.394,339.730,-98.190,174.980,31.035,155.585
C01682=1072.388,339.482,-98.154,174.977,31.030,155.584
C01683=1072.382,339.235,-98.120,174.974,31.025,155.583
C01684=1072.376,338.987,-98.086,174.970,31.020,155.582
C01685=1072.370,338.740,-98.051,174.967,31.015,155.581
C01686=1072.364,338.492,-98.016,174.963,31.010,155.580
C01687=1072.357,338.245,-97.981,174.960,31.004,155.579
C01688=1072.351,337.997,-97.947,174.957,30.999,155.579
C01689=1072.345,337.749,-97.912,174.953,30.994,155.578
C01690=1072.339,337.503,-97.878,174.949,30.989,155.577
C01691=1072.332,337.255,-97.843,174.947,30.984,155.576
C01692=1072.326,337.007,-97.809,174.943,30.979,155.575
C01693=1072.319,336.760,-97.774,174.939,30.974,155.574
C01694=1072.313,336.512,-97.740,174.937,30.969,155.573
C01695=1072.307,336.265,-97.706,174.933,30.964,155.572
C01696=1072.301,336.017,-97.671,174.929,30.959,155.571
C01697=1072.294,335.769,-97.637,174.926,30.954,155.570
C01698=1072.288,335.522,-97.602,174.923,30.949,155.569
C01699=1072.282,335.274,-97.568,174.920,30.944,155.568
C01700=1072.276,335.027,-97.534,174.916,30.939,155.567
C01701=1072.269,334.779,-97.499,174.913,30.934,155.566
C01702=1072.263,334.532,-97.465,174.910,30.929,155.565
C01703=1072.257,334.284,-97.431,174.906,30.924,155.564
C01704=1072.251,334.036,-97.397,174.903,30.919,155.564
C01705=1072.245,333.788,-97.362,174.900,30.914,155.563
C01706=1072.239,333.541,-97.328,174.896,30.909,155.562
C01707=1072.232,333.293,-97.294,174.893,30.904,155.561
C01708=1072.226,333.046,-97.260,174.890,30.899,155.560
C01709=1072.220,332.798,-97.225,174.886,30.894,155.559
C01710=1072.214,332.550,-97.191,174.883,30.890,155.558
C01711=1072.208,332.302,-97.157,174.880,30.885,155.557
C01712=1072.202,332.055,-97.123,174.876,30.880,155.556
C01713=1072.196,331.834,-97.092,174.874,30.875,155.555
C01714=1072.191,331.614,-97.062,174.871,30.871,155.555
C01715=1072.185,331.393,-97.031,174.868,30.867,155.554
C01716=1072.180,331.173,-97.001,174.864,30.862,155.553
C01717=1072.174,330.952,-96.971,174.862,30.858,155.552
C01718=1072.168,330.730,-96.941,174.859,30.854,155.551
C01719=1072.163,330.510,-96.911,174.856,30.850,155.551
C01720=1072.157,330.289,-96.880,174.853,30.845,155.550
C01721=1072.151,330.042,-96.846,174.850,30.840,155.549
C01722=1072.144,329.793,-96.813,174.846,30.836,155.548
C01723=1072.138,329.546,-96.779,174.844,30.831,155.547
C01724=1072.131,329.298,-96.745,174.840,30.826,155.546
C01725=1072.126,329.050,-96.712,174.837,30.821,155.545
C01726=1072.119,328.802,-96.677,174.834,30.817,155.545
C01727=1072.113,328.555,-96.644,174.830,30.812,155.544
C01728=1072.107,328.308,-96.610,174.827,30.807,155.543
C01729=1072.100,328.060,-96.577,174.824,30.802,155.542
C01730=1072.094,327.813,-96.543,174.820,30.797,155.541
C01731=1072.088,327.564,-96.509,174.818,30.793,155.540
C01732=1072.081,327.317,-96.475,174.814,30.788,155.539
C01733=1072.076,327.069,-96.442,174.810,30.783,155.539
C01734=1072.069,326.821,-96.408,174.808,30.779,155.538
C01735=1072.063,326.574,-96.375,174.804,30.774,155.537
C01736=1072.056,326.327,-96.341,174.802,30.769,155.536
C01737=1072.050,326.078,-96.308,174.798,30.765,155.535
C01738=1072.044,325.831,-96.274,174.795,30.760,155.534
C01739=1072.038,325.583,-96.241,174.792,30.755,155.533
C01740=1072.031,325.336,-96.208,174.788,30.750,155.533
C01741=1072.025,325.087,-96.174,174.785,30.745,155.532
C01742=1072.019,324.840,-96.140,174.782,30.741,155.531
C01743=1072.013,324.593,-96.107,174.779,30.736,155.530
C01744=1072.007,324.344,-96.073,174.775,30.732,155.529
C01745=1072.000,324.097,-96.040,174.773,30.727,155.528
C01746=1071.995,323.849,-96.007,174.769,30.722,155.527
C01747=1071.988,323.602,-95.973,174.766,30.717,155.527
C01748=1071.983,323.354,-95.940,174.763,30.712,155.526
C01749=1071.976,323.106,-95.907,174.759,30.708,155.525
C01750=1071.970,322.858,-95.873,174.757,30.703,155.524
C01751=1071.964,322.611,-95.840,174.753,30.699,155.523
C01752=1071.958,322.363,-95.806,174.750,30.694,155.522
C01753=1071.952,322.116,-95.774,174.747,30.689,155.521
C01754=1071.946,321.868,-95.741,174.744,30.684,155.521
C01755=1071.939,321.620,-95.707,174.741,30.680,155.520
C01756=1071.933,321.372,-95.674,174.738,30.675,155.519
C01757=1071.927,321.124,-95.640,174.734,30.671,155.518
C01758=1071.921,320.877,-95.608,174.732,30.666,155.517
C01759=1071.915,320.629,-95.574,174.728,30.661,155.516
C01760=1071.909,320.381,-95.542,174.725,30.657,155.516
C01761=1071.904,320.133,-95.508,174.722,30.652,155.515
C01762=1071.897,319.887,-95.475,174.719,30.648,155.514
C01763=1071.891,319.639,-95.442,174.716,30.643,155.513
C01764=1071.884,319.390,-95.408,174.713,30.638,155.512
C01765=1071.878,319.143,-95.376,174.709,30.633,155.511
C01766=1071.873,318.895,-95.342,174.707,30.629,155.511
C01767=1071.866,318.647,-95.310,174.703,30.624,155.510
C01768=1071.860,318.400,-95.277,174.701,30.620,155.509
C01769=1071.856,318.176,-95.247,174.698,30.615,155.508
C01770=1071.849,317.952,-95.217,174.694,30.611,155.507
C01771=1071.845,317.728,-95.188,174.692,30.607,155.507
C01772=1071.839,317.504,-95.157,174.689,30.603,155.506
C01773=1071.834,317.280,-95.128,174.686,30.599,155.505
C01774=1071.828,317.056,-95.099,174.684,30.595,155.504
C01775=1071.822,316.832,-95.068,174.681,30.590,155.504
C01776=1071.818,316.608,-95.039,174.678,30.587,155.503
C01777=1071.811,316.360,-95.006,174.675,30.581,155.502
C01778=1071.805,316.113,-94.973,174.672,30.577,155.501
C01779=1071.799,315.865,-94.940,174.668,30.573,155.500
C01780=1071.793,315.617,-94.907,174.666,30.568,155.500
C01781=1071.787,315.369,-94.875,174.662,30.563,155.499
C01782=1071.782,315.121,-94.842,174.660,30.559,155.498
C01783=1071.775,314.873,-94.809,174.657,30.554,155.497
C01784=1071.770,314.627,-94.777,174.653,30.550,155.496
C01785=1071.764,314.378,-94.744,174.651,30.545,155.495
C01786=1071.758,314.130,-94.711,174.647,30.541,155.495
C01787=1071.752,313.883,-94.679,174.645,30.536,155.494
C01788=1071.746,313.635,-94.647,174.641,30.532,155.493
C01789=1071.740,313.387,-94.614,174.638,30.528,155.492
C01790=1071.733,313.140,-94.582,174.635,30.523,155.492
C01791=1071.727,312.892,-94.550,174.632,30.519,155.491
C01792=1071.720,312.644,-94.517,174.629,30.514,155.490
C01793=1071.714,312.396,-94.485,174.626,30.510,155.489
C01794=1071.708,312.148,-94.452,174.623,30.506,155.488
C01795=1071.702,311.900,-94.420,174.620,30.501,155.488
